		(* Ziel												UTF8->ASCII		BacNet Text		Textlistname									BacNet Funktion																BacNet Textlist type												TextId		*)	
		I_BO_3.sActiveText								:= 	fcUtfToAscii(	fcGetBcText(	GVL_BACNET.fbBacNetParameter.metGetTextListName(enTypeOfBacNetFunktionIn := enTypeOfBacNetFunktion.Type_Anlagefunktion,		enTypeOfBacNetTextListIn := enTypeOfBacNetTextList.PRESENTVALUE	),	'I_BO_3_ST_ACTIVE'		));
		I_BO_3.sInactiveText							:= 	fcUtfToAscii(	fcGetBcText(	GVL_BACNET.fbBacNetParameter.metGetTextListName(enTypeOfBacNetFunktionIn := enTypeOfBacNetFunktion.Type_Anlagefunktion,		enTypeOfBacNetTextListIn := enTypeOfBacNetTextList.PRESENTVALUE	),	'I_BO_3_ST_INACTIVE'	));	

		(* Ziel												Convert			BacNet Text		Textlistname									BacNet Funktion																BacNet Textlist type												TextId		*)	
		I_BO_3.udiNotificationClass						:= 	TO_UDINT	(	fcGetBcText(	GVL_BACNET.fbBacNetParameter.metGetTextListName(enTypeOfBacNetFunktionIn := enTypeOfBacNetFunktion.Type_Anlagefunktion,		enTypeOfBacNetTextListIn := enTypeOfBacNetTextList.NC			),	'I_BO_3_NC'	));	
		I_BO_3.eNotifyType								:= 	WagoTypesBACnet.eBACnetNotifyType.NOTIFY_TYPE_EVENT;
		
	ELSE
		I_BO_3.Delete();
	END_IF;
	(* Get Status *)
	metCreate_I_BO_3 := I_BO_3.xIsCreated;	
END_IF;
END_METHOD

METHOD metCreate_D_BV_4 : BOOL
(* D_BV_4*)
IF NOT D_BV_4.xIsCreated THEN
	(* Ziel						UTF8->ASCII						OBJ_NAME_BASE			BacNet Text		Textlistname									BacNet Funktion																BacNet Textlist type												TextId		*)
	D_BV_4._sObjectName		:=	fcUtfToAscii(Standard.CONCAT(	OBJ_NAME_BASE		,	fcGetBcText(	GVL_BACNET.fbBacNetParameter.metGetTextListName(enTypeOfBacNetFunktionIn := enTypeOfBacNetFunktion.Type_Anlagefunktion,		enTypeOfBacNetTextListIn := enTypeOfBacNetTextList.ENDING		),	'D_BV_4')));
	D_BV_4._sDescription	:= 	fcUtfToAscii(Standard.CONCAT(	OBJ_NAME_DESCRIPTION,	fcGetBcText(	GVL_BACNET.fbBacNetParameter.metGetTextListName(enTypeOfBacNetFunktionIn := enTypeOfBacNetFunktion.Type_Anlagefunktion,		enTypeOfBacNetTextListIn := enTypeOfBacNetTextList.DESCRIPTION	),	'D_BV_4')));
	(* Create Id from Base Id and Object Nr (Last nummber of Name *)	
	D_BV_4.Create(diInstance := TO_DINT(Standard.CONCAT(TO_STRING(dwOBJ_ID_BASE),'1')));
	(* Check if Created *)
	IF D_BV_4.xIsCreated THEN
		(* Set Group *)
		D_BV_4.setPropertyGroup(WagoTypesBacNet.eBACnetPropertyIdentifier.PROP_PRESENT_VALUE						,WagoTypesBacNet.eBACnetPropertyUpdateGroup.GROUP_CYCLIC);
		D_BV_4.setPropertyGroup(WagoTypesBacNet.eBACnetPropertyIdentifier.PROP_PRIORITY_ARRAY						,WagoTypesBacNet.eBACnetPropertyUpdateGroup.GROUP_CYCLIC);
		D_BV_4.setPropertyGroup(WagoTypesBacNet.eBACnetPropertyIdentifier.PROP_ELAPSED_ACTIVE_TIME					,WagoTypesBacNet.eBACnetPropertyUpdateGroup.GROUP_CYCLIC);
		D_BV_4.setPropertyGroup(WagoTypesBacNet.eBACnetPropertyIdentifier.PROP_DESCRIPTION							,WagoTypesBacNet.eBACnetPropertyUpdateGroup.GROUP_CYCLIC);
		D_BV_4.setPropertyGroup(WagoTypesBacNet.eBACnetPropertyIdentifier.PROP_EVENT_MESSAGE_TEXTS_CONFIG			,WagoTypesBacNet.eBACnetPropertyUpdateGroup.GROUP_CYCLIC);
			
		(* Ziel												UTF8->ASCII		BacNet Text		Textlistname									BacNet Funktion																BacNet Textlist type												TextId		*)
		D_BV_4.IEventMessageTextsConfig.sToOffNormal	:=	fcUtfToAscii(	fcGetBcText(	GVL_BACNET.fbBacNetParameter.metGetTextListName(enTypeOfBacNetFunktionIn := enTypeOfBacNetFunktion.Type_Anlagefunktion,		enTypeOfBacNetTextListIn := enTypeOfBacNetTextList.EVENTMESSAGE	),	'D_BV_4_ToOffNormal'	));		
		D_BV_4.IEventMessageTextsConfig.sToFault		:=	fcUtfToAscii(	fcGetBcText(	GVL_BACNET.fbBacNetParameter.metGetTextListName(enTypeOfBacNetFunktionIn := enTypeOfBacNetFunktion.Type_Anlagefunktion,		enTypeOfBacNetTextListIn := enTypeOfBacNetTextList.EVENTMESSAGE	),	'D_BV_4_ToFault'		));		
		D_BV_4.IEventMessageTextsConfig.sToNormal		:=	fcUtfToAscii(	fcGetBcText(	GVL_BACNET.fbBacNetParameter.metGetTextListName(enTypeOfBacNetFunktionIn := enTypeOfBacNetFunktion.Type_Anlagefunktion,		enTypeOfBacNetTextListIn := enTypeOfBacNetTextList.EVENTMESSAGE	),	'D_BV_4_ToNormal'		));		

		(* Ziel												UTF8->ASCII		BacNet Text		Textlistname									BacNet Funktion																BacNet Textlist type												TextId		*)	
		D_BV_4.sActiveText								:= 	fcUtfToAscii(	fcGetBcText(	GVL_BACNET.fbBacNetParameter.metGetTextListName(enTypeOfBacNetFunktionIn := enTypeOfBacNetFunktion.Type_Anlagefunktion,		enTypeOfBacNetTextListIn := enTypeOfBacNetTextList.PRESENTVALUE	),	'D_BV_4_ST_ACTIVE'		));
		D_BV_4.sInactiveText							:= 	fcUtfToAscii(	fcGetBcText(	GVL_BACNET.fbBacNetParameter.metGetTextListName(enTypeOfBacNetFunktionIn := enTypeOfBacNetFunktion.Type_Anlagefunktion,		enTypeOfBacNetTextListIn := enTypeOfBacNetTextList.PRESENTVALUE	),	'D_BV_4_ST_INACTIVE'	));	

		(* Ziel												Convert			BacNet Text		Textlistname									BacNet Funktion																BacNet Textlist type												TextId		*)	
		D_BV_4.udiNotificationClass						:= 	TO_UDINT	(	fcGetBcText(	GVL_BACNET.fbBacNetParameter.metGetTextListName(enTypeOfBacNetFunktionIn := enTypeOfBacNetFunktion.Type_Anlagefunktion,		enTypeOfBacNetTextListIn := enTypeOfBacNetTextList.NC			),	'D_BV_4_NC'	));	
		D_BV_4.eNotifyType								:= 	WagoTypesBACnet.eBACnetNotifyType.NOTIFY_TYPE_EVENT;
		D_BV_4.xAlarmValue								:= 	TO_BOOL		(	fcGetBcText(	GVL_BACNET.fbBacNetParameter.metGetTextListName(enTypeOfBacNetFunktionIn := enTypeOfBacNetFunktion.Type_Anlagefunktion,		enTypeOfBacNetTextListIn := enTypeOfBacNetTextList.NC		),	'D_BV_4_ALV'	));
	ELSE
		D_BV_4.Delete();
	END_IF;
	(* Get Status *)
	metCreate_D_BV_4 := D_BV_4.xIsCreated;	
END_IF;
END_METHOD

METHOD metCreate_E_BI_1 : BOOL
(* E_BI_1*)
IF NOT E_BI_1.xIsCreated THEN
	(* Ziel						UTF8->ASCII						OBJ_NAME_BASE			BacNet Text		Textlistname									BacNet Funktion																BacNet Textlist type												TextId		*)
	E_BI_1._sObjectName		:=	fcUtfToAscii(Standard.CONCAT(	OBJ_NAME_BASE		,	fcGetBcText(	GVL_BACNET.fbBacNetParameter.metGetTextListName(enTypeOfBacNetFunktionIn := enTypeOfBacNetFunktion.Type_Anlagefunktion,		enTypeOfBacNetTextListIn := enTypeOfBacNetTextList.ENDING		),	'E_BI_1')));
	E_BI_1._sDescription	:= 	fcUtfToAscii(Standard.CONCAT(	OBJ_NAME_DESCRIPTION,	fcGetBcText(	GVL_BACNET.fbBacNetParameter.metGetTextListName(enTypeOfBacNetFunktionIn := enTypeOfBacNetFunktion.Type_Anlagefunktion,		enTypeOfBacNetTextListIn := enTypeOfBacNetTextList.DESCRIPTION	),	'E_BI_1')));
	(* Create Id from Base Id and Object Nr (Last nummber of Name *)	
	E_BI_1.Create(diInstance := TO_DINT(Standard.CONCAT(TO_STRING(dwOBJ_ID_BASE),'1')));
	(* Check if Created *)
	IF E_BI_1.xIsCreated THEN
		(* Set Group *)
		E_BI_1.setPropertyGroup(WagoTypesBacNet.eBACnetPropertyIdentifier.PROP_PRESENT_VALUE						,WagoTypesBacNet.eBACnetPropertyUpdateGroup.GROUP_CYCLIC);
		E_BI_1.setPropertyGroup(WagoTypesBacNet.eBACnetPropertyIdentifier.PROP_PRIORITY_ARRAY						,WagoTypesBacNet.eBACnetPropertyUpdateGroup.GROUP_CYCLIC);
		E_BI_1.setPropertyGroup(WagoTypesBacNet.eBACnetPropertyIdentifier.PROP_ELAPSED_ACTIVE_TIME					,WagoTypesBacNet.eBACnetPropertyUpdateGroup.GROUP_CYCLIC);
		E_BI_1.setPropertyGroup(WagoTypesBacNet.eBACnetPropertyIdentifier.PROP_DESCRIPTION							,WagoTypesBacNet.eBACnetPropertyUpdateGroup.GROUP_CYCLIC);
		E_BI_1.setPropertyGroup(WagoTypesBacNet.eBACnetPropertyIdentifier.PROP_EVENT_MESSAGE_TEXTS_CONFIG			,WagoTypesBacNet.eBACnetPropertyUpdateGroup.GROUP_CYCLIC);
			
		(* Ziel												UTF8->ASCII		BacNet Text		Textlistname									BacNet Funktion																BacNet Textlist type												TextId		*)
		E_BI_1.IEventMessageTextsConfig.sToOffNormal	:=	fcUtfToAscii(	fcGetBcText(	GVL_BACNET.fbBacNetParameter.metGetTextListName(enTypeOfBacNetFunktionIn := enTypeOfBacNetFunktion.Type_Anlagefunktion,		enTypeOfBacNetTextListIn := enTypeOfBacNetTextList.EVENTMESSAGE	),	'E_BI_1_ToOffNormal'	));		
		E_BI_1.IEventMessageTextsConfig.sToFault		:=	fcUtfToAscii(	fcGetBcText(	GVL_BACNET.fbBacNetParameter.metGetTextListName(enTypeOfBacNetFunktionIn := enTypeOfBacNetFunktion.Type_Anlagefunktion,		enTypeOfBacNetTextListIn := enTypeOfBacNetTextList.EVENTMESSAGE	),	'E_BI_1_ToFault'		));		
		E_BI_1.IEventMessageTextsConfig.sToNormal		:=	fcUtfToAscii(	fcGetBcText(	GVL_BACNET.fbBacNetParameter.metGetTextListName(enTypeOfBacNetFunktionIn := enTypeOfBacNetFunktion.Type_Anlagefunktion,		enTypeOfBacNetTextListIn := enTypeOfBacNetTextList.EVENTMESSAGE	),	'E_BI_1_ToNormal'		));		

		(* Ziel												UTF8->ASCII		BacNet Text		Textlistname									BacNet Funktion																BacNet Textlist type												TextId		*)	
		E_BI_1.sActiveText								:= 	fcUtfToAscii(	fcGetBcText(	GVL_BACNET.fbBacNetParameter.metGetTextListName(enTypeOfBacNetFunktionIn := enTypeOfBacNetFunktion.Type_Anlagefunktion,		enTypeOfBacNetTextListIn := enTypeOfBacNetTextList.PRESENTVALUE	),	'E_BI_1_ST_ACTIVE'		));
		E_BI_1.sInactiveText							:= 	fcUtfToAscii(	fcGetBcText(	GVL_BACNET.fbBacNetParameter.metGetTextListName(enTypeOfBacNetFunktionIn := enTypeOfBacNetFunktion.Type_Anlagefunktion,		enTypeOfBacNetTextListIn := enTypeOfBacNetTextList.PRESENTVALUE	),	'E_BI_1_ST_INACTIVE'	));	

		(* Ziel												Convert			BacNet Text		Textlistname									BacNet Funktion																BacNet Textlist type												TextId		*)	
		E_BI_1.udiNotificationClass						:= 	TO_UDINT	(	fcGetBcText(	GVL_BACNET.fbBacNetParameter.metGetTextListName(enTypeOfBacNetFunktionIn := enTypeOfBacNetFunktion.Type_Anlagefunktion,		enTypeOfBacNetTextListIn := enTypeOfBacNetTextList.NC			),	'E_BI_1_NC'	));	
		E_BI_1.eNotifyType								:= 	WagoTypesBACnet.eBACnetNotifyType.NOTIFY_TYPE_EVENT;
		E_BI_1.xAlarmValue								:= 	TO_BOOL		(	fcGetBcText(	GVL_BACNET.fbBacNetParameter.metGetTextListName(enTypeOfBacNetFunktionIn := enTypeOfBacNetFunktion.Type_Anlagefunktion,		enTypeOfBacNetTextListIn := enTypeOfBacNetTextList.NC			),	'E_BI_1_ALV'	));
	ELSE
		E_BI_1.Delete();
	END_IF;
	(* Get Status *)
	metCreate_E_BI_1 := E_BI_1.xIsCreated;	
END_IF;
END_METHOD

METHOD metCreate_B_BV_2 : BOOL
(* B_BV_2*)
IF NOT B_BV_2.xIsCreated THEN
	(* Ziel						UTF8->ASCII						OBJ_NAME_BASE			BacNet Text		Textlistname									BacNet Funktion																BacNet Textlist type												TextId		*)
	B_BV_2._sObjectName		:=	fcUtfToAscii(Standard.CONCAT(	OBJ_NAME_BASE		,	fcGetBcText(	GVL_BACNET.fbBacNetParameter.metGetTextListName(enTypeOfBacNetFunktionIn := enTypeOfBacNetFunktion.Type_Anlagefunktion,		enTypeOfBacNetTextListIn := enTypeOfBacNetTextList.ENDING		),	'B_BV_2')));
	B_BV_2._sDescription	:= 	fcUtfToAscii(Standard.CONCAT(	OBJ_NAME_DESCRIPTION,	fcGetBcText(	GVL_BACNET.fbBacNetParameter.metGetTextListName(enTypeOfBacNetFunktionIn := enTypeOfBacNetFunktion.Type_Anlagefunktion,		enTypeOfBacNetTextListIn := enTypeOfBacNetTextList.DESCRIPTION	),	'B_BV_2')));
	(* Create Id from Base Id and Object Nr (Last nummber of Name *)	
	B_BV_2.Create(diInstance := TO_DINT(Standard.CONCAT(TO_STRING(dwOBJ_ID_BASE),'1')));
	(* Check if Created *)
	IF B_BV_2.xIsCreated THEN
		(* Set Group *)
		B_BV_2.setPropertyGroup(WagoTypesBacNet.eBACnetPropertyIdentifier.PROP_PRESENT_VALUE						,WagoTypesBacNet.eBACnetPropertyUpdateGroup.GROUP_CYCLIC);
		B_BV_2.setPropertyGroup(WagoTypesBacNet.eBACnetPropertyIdentifier.PROP_PRIORITY_ARRAY						,WagoTypesBacNet.eBACnetPropertyUpdateGroup.GROUP_CYCLIC);
		B_BV_2.setPropertyGroup(WagoTypesBacNet.eBACnetPropertyIdentifier.PROP_ELAPSED_ACTIVE_TIME					,WagoTypesBacNet.eBACnetPropertyUpdateGroup.GROUP_CYCLIC);
		B_BV_2.setPropertyGroup(WagoTypesBacNet.eBACnetPropertyIdentifier.PROP_DESCRIPTION							,WagoTypesBacNet.eBACnetPropertyUpdateGroup.GROUP_CYCLIC);
		B_BV_2.setPropertyGroup(WagoTypesBacNet.eBACnetPropertyIdentifier.PROP_EVENT_MESSAGE_TEXTS_CONFIG			,WagoTypesBacNet.eBACnetPropertyUpdateGroup.GROUP_CYCLIC);
			
		(* Ziel												UTF8->ASCII		BacNet Text		Textlistname									BacNet Funktion																BacNet Textlist type												TextId		*)
		B_BV_2.IEventMessageTextsConfig.sToOffNormal	:=	fcUtfToAscii(	fcGetBcText(	GVL_BACNET.fbBacNetParameter.metGetTextListName(enTypeOfBacNetFunktionIn := enTypeOfBacNetFunktion.Type_Anlagefunktion,		enTypeOfBacNetTextListIn := enTypeOfBacNetTextList.EVENTMESSAGE	),	'B_BV_2_ToOffNormal'	));		
		B_BV_2.IEventMessageTextsConfig.sToFault		:=	fcUtfToAscii(	fcGetBcText(	GVL_BACNET.fbBacNetParameter.metGetTextListName(enTypeOfBacNetFunktionIn := enTypeOfBacNetFunktion.Type_Anlagefunktion,		enTypeOfBacNetTextListIn := enTypeOfBacNetTextList.EVENTMESSAGE	),	'B_BV_2_ToFault'		));		
		B_BV_2.IEventMessageTextsConfig.sToNormal		:=	fcUtfToAscii(	fcGetBcText(	GVL_BACNET.fbBacNetParameter.metGetTextListName(enTypeOfBacNetFunktionIn := enTypeOfBacNetFunktion.Type_Anlagefunktion,		enTypeOfBacNetTextListIn := enTypeOfBacNetTextList.EVENTMESSAGE	),	'B_BV_2_ToNormal'		));		

		(* Ziel												UTF8->ASCII		BacNet Text		Textlistname									BacNet Funktion																BacNet Textlist type												TextId		*)	
		B_BV_2.sActiveText								:= 	fcUtfToAscii(	fcGetBcText(	GVL_BACNET.fbBacNetParameter.metGetTextListName(enTypeOfBacNetFunktionIn := enTypeOfBacNetFunktion.Type_Anlagefunktion,		enTypeOfBacNetTextListIn := enTypeOfBacNetTextList.PRESENTVALUE	),	'B_BV_2_ST_ACTIVE'		));
		B_BV_2.sInactiveText							:= 	fcUtfToAscii(	fcGetBcText(	GVL_BACNET.fbBacNetParameter.metGetTextListName(enTypeOfBacNetFunktionIn := enTypeOfBacNetFunktion.Type_Anlagefunktion,		enTypeOfBacNetTextListIn := enTypeOfBacNetTextList.PRESENTVALUE	),	'B_BV_2_ST_INACTIVE'	));	

		(* Ziel												Convert			BacNet Text		Textlistname									BacNet Funktion																BacNet Textlist type												TextId		*)	
		B_BV_2.udiNotificationClass						:= 	TO_UDINT	(	fcGetBcText(	GVL_BACNET.fbBacNetParameter.metGetTextListName(enTypeOfBacNetFunktionIn := enTypeOfBacNetFunktion.Type_Anlagefunktion,		enTypeOfBacNetTextListIn := enTypeOfBacNetTextList.NC			),	'B_BV_2_NC'	));	
		B_BV_2.eNotifyType								:= 	WagoTypesBACnet.eBACnetNotifyType.NOTIFY_TYPE_ALARM;
		B_BV_2.xAlarmValue								:= 	TO_BOOL		(	fcGetBcText(	GVL_BACNET.fbBacNetParameter.metGetTextListName(enTypeOfBacNetFunktionIn := enTypeOfBacNetFunktion.Type_Anlagefunktion,		enTypeOfBacNetTextListIn := enTypeOfBacNetTextList.NC		),	'B_BV_2_ALV'	));
		
	ELSE
		B_BV_2.Delete();
	END_IF;
	(* Get Status *)
	metCreate_B_BV_2 := B_BV_2.xIsCreated;	
END_IF;
END_METHOD

METHOD metCreate_C_BV_3 : BOOL
(* C_BV_3*)
IF NOT C_BV_3.xIsCreated THEN
	(* Ziel						UTF8->ASCII						OBJ_NAME_BASE			BacNet Text		Textlistname									BacNet Funktion																BacNet Textlist type												TextId		*)
	C_BV_3._sObjectName		:=	fcUtfToAscii(Standard.CONCAT(	OBJ_NAME_BASE		,	fcGetBcText(	GVL_BACNET.fbBacNetParameter.metGetTextListName(enTypeOfBacNetFunktionIn := enTypeOfBacNetFunktion.Type_Anlagefunktion,		enTypeOfBacNetTextListIn := enTypeOfBacNetTextList.ENDING		),	'C_BV_3')));
	C_BV_3._sDescription	:= 	fcUtfToAscii(Standard.CONCAT(	OBJ_NAME_DESCRIPTION,	fcGetBcText(	GVL_BACNET.fbBacNetParameter.metGetTextListName(enTypeOfBacNetFunktionIn := enTypeOfBacNetFunktion.Type_Anlagefunktion,		enTypeOfBacNetTextListIn := enTypeOfBacNetTextList.DESCRIPTION	),	'C_BV_3')));
	(* Create Id from Base Id and Object Nr (Last nummber of Name *)	
	C_BV_3.Create(diInstance := TO_DINT(Standard.CONCAT(TO_STRING(dwOBJ_ID_BASE),'1')));
	(* Check if Created *)
	IF C_BV_3.xIsCreated THEN
		(* Set Group *)
		C_BV_3.setPropertyGroup(WagoTypesBacNet.eBACnetPropertyIdentifier.PROP_PRESENT_VALUE						,WagoTypesBacNet.eBACnetPropertyUpdateGroup.GROUP_CYCLIC);
		C_BV_3.setPropertyGroup(WagoTypesBacNet.eBACnetPropertyIdentifier.PROP_PRIORITY_ARRAY						,WagoTypesBacNet.eBACnetPropertyUpdateGroup.GROUP_CYCLIC);
		C_BV_3.setPropertyGroup(WagoTypesBacNet.eBACnetPropertyIdentifier.PROP_ELAPSED_ACTIVE_TIME					,WagoTypesBacNet.eBACnetPropertyUpdateGroup.GROUP_CYCLIC);
		C_BV_3.setPropertyGroup(WagoTypesBacNet.eBACnetPropertyIdentifier.PROP_DESCRIPTION							,WagoTypesBacNet.eBACnetPropertyUpdateGroup.GROUP_CYCLIC);
		C_BV_3.setPropertyGroup(WagoTypesBacNet.eBACnetPropertyIdentifier.PROP_EVENT_MESSAGE_TEXTS_CONFIG			,WagoTypesBacNet.eBACnetPropertyUpdateGroup.GROUP_CYCLIC);
			
		(* Ziel												UTF8->ASCII		BacNet Text		Textlistname									BacNet Funktion																BacNet Textlist type												TextId		*)
		C_BV_3.IEventMessageTextsConfig.sToOffNormal	:=	fcUtfToAscii(	fcGetBcText(	GVL_BACNET.fbBacNetParameter.metGetTextListName(enTypeOfBacNetFunktionIn := enTypeOfBacNetFunktion.Type_Anlagefunktion,		enTypeOfBacNetTextListIn := enTypeOfBacNetTextList.EVENTMESSAGE	),	'C_BV_3_ToOffNormal'	));		
		C_BV_3.IEventMessageTextsConfig.sToFault		:=	fcUtfToAscii(	fcGetBcText(	GVL_BACNET.fbBacNetParameter.metGetTextListName(enTypeOfBacNetFunktionIn := enTypeOfBacNetFunktion.Type_Anlagefunktion,		enTypeOfBacNetTextListIn := enTypeOfBacNetTextList.EVENTMESSAGE	),	'C_BV_3_ToFault'		));		
		C_BV_3.IEventMessageTextsConfig.sToNormal		:=	fcUtfToAscii(	fcGetBcText(	GVL_BACNET.fbBacNetParameter.metGetTextListName(enTypeOfBacNetFunktionIn := enTypeOfBacNetFunktion.Type_Anlagefunktion,		enTypeOfBacNetTextListIn := enTypeOfBacNetTextList.EVENTMESSAGE	),	'C_BV_3_ToNormal'		));		

		(* Ziel												UTF8->ASCII		BacNet Text		Textlistname									BacNet Funktion																BacNet Textlist type												TextId		*)	
		C_BV_3.sActiveText								:= 	fcUtfToAscii(	fcGetBcText(	GVL_BACNET.fbBacNetParameter.metGetTextListName(enTypeOfBacNetFunktionIn := enTypeOfBacNetFunktion.Type_Anlagefunktion,		enTypeOfBacNetTextListIn := enTypeOfBacNetTextList.PRESENTVALUE	),	'C_BV_3_ST_ACTIVE'		));
		C_BV_3.sInactiveText							:= 	fcUtfToAscii(	fcGetBcText(	GVL_BACNET.fbBacNetParameter.metGetTextListName(enTypeOfBacNetFunktionIn := enTypeOfBacNetFunktion.Type_Anlagefunktion,		enTypeOfBacNetTextListIn := enTypeOfBacNetTextList.PRESENTVALUE	),	'C_BV_3_ST_INACTIVE'	));	

		(* Ziel												Convert			BacNet Text		Textlistname									BacNet Funktion																BacNet Textlist type												TextId		*)	
		C_BV_3.udiNotificationClass						:= 	TO_UDINT	(	fcGetBcText(	GVL_BACNET.fbBacNetParameter.metGetTextListName(enTypeOfBacNetFunktionIn := enTypeOfBacNetFunktion.Type_Anlagefunktion,		enTypeOfBacNetTextListIn := enTypeOfBacNetTextList.NC			),	'C_BV_3_NC'	));	
		C_BV_3.eNotifyType								:= 	WagoTypesBACnet.eBACnetNotifyType.NOTIFY_TYPE_ALARM;
		C_BV_3.xAlarmValue								:= 	TO_BOOL		(	fcGetBcText(	GVL_BACNET.fbBacNetParameter.metGetTextListName(enTypeOfBacNetFunktionIn := enTypeOfBacNetFunktion.Type_Anlagefunktion,		enTypeOfBacNetTextListIn := enTypeOfBacNetTextList.NC		),	'C_BV_3_ALV'	));
	ELSE
		C_BV_3.Delete();
	END_IF;
	(* Get Status *)
	metCreate_C_BV_3 := C_BV_3.xIsCreated;	
END_IF;
END_METHOD

METHOD metCreate_J_SC_1 : BOOL
(* J_SC_1*)
IF NOT J_SC_1.xIsCreated THEN
	(* Ziel						UTF8->ASCII						OBJ_NAME_BASE			BacNet Text		Textlistname									BacNet Funktion																BacNet Textlist type												TextId		*)
	J_SC_1._sObjectName		:=	fcUtfToAscii(Standard.CONCAT(	OBJ_NAME_BASE		,	fcGetBcText(	GVL_BACNET.fbBacNetParameter.metGetTextListName(enTypeOfBacNetFunktionIn := enTypeOfBacNetFunktion.Type_Anlagefunktion,		enTypeOfBacNetTextListIn := enTypeOfBacNetTextList.ENDING		),	'J_SC_1')));
	J_SC_1._sDescription	:= 	fcUtfToAscii(Standard.CONCAT(	OBJ_NAME_DESCRIPTION,	fcGetBcText(	GVL_BACNET.fbBacNetParameter.metGetTextListName(enTypeOfBacNetFunktionIn := enTypeOfBacNetFunktion.Type_Anlagefunktion,		enTypeOfBacNetTextListIn := enTypeOfBacNetTextList.DESCRIPTION	),	'J_SC_1')));
	(* Create Id from Base Id and Object Nr (Last nummber of Name *)	
	J_SC_1.Create(diInstance := TO_DINT(Standard.CONCAT(TO_STRING(dwOBJ_ID_BASE),'1')));
	(* Check if Created *)
	IF J_SC_1.xIsCreated THEN
		(* Set Group *)
		J_SC_1.setPropertyGroup(WagoTypesBacNet.eBACnetPropertyIdentifier.PROP_PRESENT_VALUE						,WagoTypesBacNet.eBACnetPropertyUpdateGroup.GROUP_CYCLIC);
		J_SC_1.setPropertyGroup(WagoTypesBacNet.eBACnetPropertyIdentifier.PROP_PRIORITY_ARRAY						,WagoTypesBacNet.eBACnetPropertyUpdateGroup.GROUP_CYCLIC);
		J_SC_1.setPropertyGroup(WagoTypesBacNet.eBACnetPropertyIdentifier.PROP_ELAPSED_ACTIVE_TIME					,WagoTypesBacNet.eBACnetPropertyUpdateGroup.GROUP_CYCLIC);
		J_SC_1.setPropertyGroup(WagoTypesBacNet.eBACnetPropertyIdentifier.PROP_DESCRIPTION							,WagoTypesBacNet.eBACnetPropertyUpdateGroup.GROUP_CYCLIC);
		J_SC_1.setPropertyGroup(WagoTypesBacNet.eBACnetPropertyIdentifier.PROP_EVENT_MESSAGE_TEXTS_CONFIG			,WagoTypesBacNet.eBACnetPropertyUpdateGroup.GROUP_CYCLIC);
			
		(* Ziel												UTF8->ASCII		BacNet Text		Textlistname									BacNet Funktion																BacNet Textlist type												TextId		*)
		J_SC_1.IEventMessageTextsConfig.sToOffNormal	:=	fcUtfToAscii(	fcGetBcText(	GVL_BACNET.fbBacNetParameter.metGetTextListName(enTypeOfBacNetFunktionIn := enTypeOfBacNetFunktion.Type_Anlagefunktion,		enTypeOfBacNetTextListIn := enTypeOfBacNetTextList.EVENTMESSAGE	),	'J_SC_1_ToOffNormal'	));		
		J_SC_1.IEventMessageTextsConfig.sToFault		:=	fcUtfToAscii(	fcGetBcText(	GVL_BACNET.fbBacNetParameter.metGetTextListName(enTypeOfBacNetFunktionIn := enTypeOfBacNetFunktion.Type_Anlagefunktion,		enTypeOfBacNetTextListIn := enTypeOfBacNetTextList.EVENTMESSAGE	),	'J_SC_1_ToFault'		));		
		J_SC_1.IEventMessageTextsConfig.sToNormal		:=	fcUtfToAscii(	fcGetBcText(	GVL_BACNET.fbBacNetParameter.metGetTextListName(enTypeOfBacNetFunktionIn := enTypeOfBacNetFunktion.Type_Anlagefunktion,		enTypeOfBacNetTextListIn := enTypeOfBacNetTextList.EVENTMESSAGE	),	'J_SC_1_ToNormal'		));		

		(* Ziel												Convert			BacNet Text		Textlistname									BacNet Funktion																BacNet Textlist type												TextId		*)	
		J_SC_1.udiNotificationClass						:= 	TO_UDINT	(	fcGetBcText(	GVL_BACNET.fbBacNetParameter.metGetTextListName(enTypeOfBacNetFunktionIn := enTypeOfBacNetFunktion.Type_Anlagefunktion,		enTypeOfBacNetTextListIn := enTypeOfBacNetTextList.NC			),	'J_SC_1_NC'	));	
		J_SC_1.eNotifyType								:= 	WagoTypesBACnet.eBACnetNotifyType.NOTIFY_TYPE_EVENT;
		
	ELSE
		J_SC_1.Delete();
	END_IF;
	(* Get Status *)
	metCreate_J_SC_1 := J_SC_1.xIsCreated;	
END_IF;
END_METHOD

METHOD metCreate_F_BV_5 : BOOL
(* F_BV_5*)
IF NOT F_BV_5.xIsCreated THEN
	(* Ziel						UTF8->ASCII						OBJ_NAME_BASE			BacNet Text		Textlistname									BacNet Funktion																BacNet Textlist type												TextId		*)
	F_BV_5._sObjectName		:=	fcUtfToAscii(Standard.CONCAT(	OBJ_NAME_BASE		,	fcGetBcText(	GVL_BACNET.fbBacNetParameter.metGetTextListName(enTypeOfBacNetFunktionIn := enTypeOfBacNetFunktion.Type_Anlagefunktion,		enTypeOfBacNetTextListIn := enTypeOfBacNetTextList.ENDING		),	'F_BV_5')));
	F_BV_5._sDescription	:= 	fcUtfToAscii(Standard.CONCAT(	OBJ_NAME_DESCRIPTION,	fcGetBcText(	GVL_BACNET.fbBacNetParameter.metGetTextListName(enTypeOfBacNetFunktionIn := enTypeOfBacNetFunktion.Type_Anlagefunktion,		enTypeOfBacNetTextListIn := enTypeOfBacNetTextList.DESCRIPTION	),	'F_BV_5')));
	(* Create Id from Base Id and Object Nr (Last nummber of Name *)	
	F_BV_5.Create(diInstance := TO_DINT(Standard.CONCAT(TO_STRING(dwOBJ_ID_BASE),'1')));
	(* Check if Created *)
	IF F_BV_5.xIsCreated THEN
		(* Set Group *)
		F_BV_5.setPropertyGroup(WagoTypesBacNet.eBACnetPropertyIdentifier.PROP_PRESENT_VALUE						,WagoTypesBacNet.eBACnetPropertyUpdateGroup.GROUP_CYCLIC);
		F_BV_5.setPropertyGroup(WagoTypesBacNet.eBACnetPropertyIdentifier.PROP_PRIORITY_ARRAY						,WagoTypesBacNet.eBACnetPropertyUpdateGroup.GROUP_CYCLIC);
		F_BV_5.setPropertyGroup(WagoTypesBacNet.eBACnetPropertyIdentifier.PROP_ELAPSED_ACTIVE_TIME					,WagoTypesBacNet.eBACnetPropertyUpdateGroup.GROUP_CYCLIC);
		F_BV_5.setPropertyGroup(WagoTypesBacNet.eBACnetPropertyIdentifier.PROP_DESCRIPTION							,WagoTypesBacNet.eBACnetPropertyUpdateGroup.GROUP_CYCLIC);
		F_BV_5.setPropertyGroup(WagoTypesBacNet.eBACnetPropertyIdentifier.PROP_EVENT_MESSAGE_TEXTS_CONFIG			,WagoTypesBacNet.eBACnetPropertyUpdateGroup.GROUP_CYCLIC);
			
		(* Ziel												UTF8->ASCII		BacNet Text		Textlistname									BacNet Funktion																BacNet Textlist type												TextId		*)
		F_BV_5.IEventMessageTextsConfig.sToOffNormal	:=	fcUtfToAscii(	fcGetBcText(	GVL_BACNET.fbBacNetParameter.metGetTextListName(enTypeOfBacNetFunktionIn := enTypeOfBacNetFunktion.Type_Anlagefunktion,		enTypeOfBacNetTextListIn := enTypeOfBacNetTextList.EVENTMESSAGE	),	'F_BV_5_ToOffNormal'	));		
		F_BV_5.IEventMessageTextsConfig.sToFault		:=	fcUtfToAscii(	fcGetBcText(	GVL_BACNET.fbBacNetParameter.metGetTextListName(enTypeOfBacNetFunktionIn := enTypeOfBacNetFunktion.Type_Anlagefunktion,		enTypeOfBacNetTextListIn := enTypeOfBacNetTextList.EVENTMESSAGE	),	'F_BV_5_ToFault'		));		
		F_BV_5.IEventMessageTextsConfig.sToNormal		:=	fcUtfToAscii(	fcGetBcText(	GVL_BACNET.fbBacNetParameter.metGetTextListName(enTypeOfBacNetFunktionIn := enTypeOfBacNetFunktion.Type_Anlagefunktion,		enTypeOfBacNetTextListIn := enTypeOfBacNetTextList.EVENTMESSAGE	),	'F_BV_5_ToNormal'		));		

		(* Ziel												UTF8->ASCII		BacNet Text		Textlistname									BacNet Funktion																BacNet Textlist type												TextId		*)	
		F_BV_5.sActiveText								:= 	fcUtfToAscii(	fcGetBcText(	GVL_BACNET.fbBacNetParameter.metGetTextListName(enTypeOfBacNetFunktionIn := enTypeOfBacNetFunktion.Type_Anlagefunktion,		enTypeOfBacNetTextListIn := enTypeOfBacNetTextList.PRESENTVALUE	),	'F_BV_5_ST_ACTIVE'		));
		F_BV_5.sInactiveText							:= 	fcUtfToAscii(	fcGetBcText(	GVL_BACNET.fbBacNetParameter.metGetTextListName(enTypeOfBacNetFunktionIn := enTypeOfBacNetFunktion.Type_Anlagefunktion,		enTypeOfBacNetTextListIn := enTypeOfBacNetTextList.PRESENTVALUE	),	'F_BV_5_ST_INACTIVE'	));	

		(* Ziel												Convert			BacNet Text		Textlistname									BacNet Funktion																BacNet Textlist type												TextId		*)	
		F_BV_5.udiNotificationClass						:= 	TO_UDINT	(	fcGetBcText(	GVL_BACNET.fbBacNetParameter.metGetTextListName(enTypeOfBacNetFunktionIn := enTypeOfBacNetFunktion.Type_Anlagefunktion,		enTypeOfBacNetTextListIn := enTypeOfBacNetTextList.NC			),	'F_BV_5_NC'	));	
		F_BV_5.eNotifyType								:= 	WagoTypesBACnet.eBACnetNotifyType.NOTIFY_TYPE_EVENT;
		F_BV_5.xAlarmValue								:= 	TO_BOOL		(	fcGetBcText(	GVL_BACNET.fbBacNetParameter.metGetTextListName(enTypeOfBacNetFunktionIn := enTypeOfBacNetFunktion.Type_Anlagefunktion,		enTypeOfBacNetTextListIn := enTypeOfBacNetTextList.NC			),	'F_BV_5_ALV'	));
		
	ELSE
		F_BV_5.Delete();
	END_IF;
	(* Get Status *)
	metCreate_F_BV_5 := F_BV_5.xIsCreated;	
END_IF;
END_METHOD

METHOD metCreate_G_BO_1 : BOOL
(* G_BO_1*)
IF NOT G_BO_1.xIsCreated THEN
	(* Ziel						UTF8->ASCII						OBJ_NAME_BASE			BacNet Text		Textlistname									BacNet Funktion																BacNet Textlist type												TextId		*)
	G_BO_1._sObjectName		:=	fcUtfToAscii(Standard.CONCAT(	OBJ_NAME_BASE		,	fcGetBcText(	GVL_BACNET.fbBacNetParameter.metGetTextListName(enTypeOfBacNetFunktionIn := enTypeOfBacNetFunktion.Type_Anlagefunktion,		enTypeOfBacNetTextListIn := enTypeOfBacNetTextList.ENDING		),	'G_BO_1')));
	G_BO_1._sDescription	:= 	fcUtfToAscii(Standard.CONCAT(	OBJ_NAME_DESCRIPTION,	fcGetBcText(	GVL_BACNET.fbBacNetParameter.metGetTextListName(enTypeOfBacNetFunktionIn := enTypeOfBacNetFunktion.Type_Anlagefunktion,		enTypeOfBacNetTextListIn := enTypeOfBacNetTextList.DESCRIPTION	),	'G_BO_1')));
	(* Create Id from Base Id and Object Nr (Last nummber of Name *)	
	G_BO_1.Create(diInstance := TO_DINT(Standard.CONCAT(TO_STRING(dwOBJ_ID_BASE),'1')));
	(* Check if Created *)
	IF G_BO_1.xIsCreated THEN
		(* Set Group *)
		G_BO_1.setPropertyGroup(WagoTypesBacNet.eBACnetPropertyIdentifier.PROP_PRESENT_VALUE						,WagoTypesBacNet.eBACnetPropertyUpdateGroup.GROUP_CYCLIC);
		G_BO_1.setPropertyGroup(WagoTypesBacNet.eBACnetPropertyIdentifier.PROP_PRIORITY_ARRAY						,WagoTypesBacNet.eBACnetPropertyUpdateGroup.GROUP_CYCLIC);
		G_BO_1.setPropertyGroup(WagoTypesBacNet.eBACnetPropertyIdentifier.PROP_ELAPSED_ACTIVE_TIME					,WagoTypesBacNet.eBACnetPropertyUpdateGroup.GROUP_CYCLIC);
		G_BO_1.setPropertyGroup(WagoTypesBacNet.eBACnetPropertyIdentifier.PROP_DESCRIPTION							,WagoTypesBacNet.eBACnetPropertyUpdateGroup.GROUP_CYCLIC);
		G_BO_1.setPropertyGroup(WagoTypesBacNet.eBACnetPropertyIdentifier.PROP_EVENT_MESSAGE_TEXTS_CONFIG			,WagoTypesBacNet.eBACnetPropertyUpdateGroup.GROUP_CYCLIC);
			
		(* Ziel												UTF8->ASCII		BacNet Text		Textlistname									BacNet Funktion																BacNet Textlist type												TextId		*)
		G_BO_1.IEventMessageTextsConfig.sToOffNormal	:=	fcUtfToAscii(	fcGetBcText(	GVL_BACNET.fbBacNetParameter.metGetTextListName(enTypeOfBacNetFunktionIn := enTypeOfBacNetFunktion.Type_Anlagefunktion,		enTypeOfBacNetTextListIn := enTypeOfBacNetTextList.EVENTMESSAGE	),	'G_BO_1_ToOffNormal'	));		
		G_BO_1.IEventMessageTextsConfig.sToFault		:=	fcUtfToAscii(	fcGetBcText(	GVL_BACNET.fbBacNetParameter.metGetTextListName(enTypeOfBacNetFunktionIn := enTypeOfBacNetFunktion.Type_Anlagefunktion,		enTypeOfBacNetTextListIn := enTypeOfBacNetTextList.EVENTMESSAGE	),	'G_BO_1_ToFault'		));		
		G_BO_1.IEventMessageTextsConfig.sToNormal		:=	fcUtfToAscii(	fcGetBcText(	GVL_BACNET.fbBacNetParameter.metGetTextListName(enTypeOfBacNetFunktionIn := enTypeOfBacNetFunktion.Type_Anlagefunktion,		enTypeOfBacNetTextListIn := enTypeOfBacNetTextList.EVENTMESSAGE	),	'G_BO_1_ToNormal'		));		

		(* Ziel												UTF8->ASCII		BacNet Text		Textlistname									BacNet Funktion																BacNet Textlist type												TextId		*)	
		G_BO_1.sActiveText								:= 	fcUtfToAscii(	fcGetBcText(	GVL_BACNET.fbBacNetParameter.metGetTextListName(enTypeOfBacNetFunktionIn := enTypeOfBacNetFunktion.Type_Anlagefunktion,		enTypeOfBacNetTextListIn := enTypeOfBacNetTextList.PRESENTVALUE	),	'G_BO_1_ST_ACTIVE'		));
		G_BO_1.sInactiveText							:= 	fcUtfToAscii(	fcGetBcText(	GVL_BACNET.fbBacNetParameter.metGetTextListName(enTypeOfBacNetFunktionIn := enTypeOfBacNetFunktion.Type_Anlagefunktion,		enTypeOfBacNetTextListIn := enTypeOfBacNetTextList.PRESENTVALUE	),	'G_BO_1_ST_INACTIVE'	));	

		(* Ziel												Convert			BacNet Text		Textlistname									BacNet Funktion																BacNet Textlist type												TextId		*)	
		G_BO_1.udiNotificationClass						:= 	TO_UDINT	(	fcGetBcText(	GVL_BACNET.fbBacNetParameter.metGetTextListName(enTypeOfBacNetFunktionIn := enTypeOfBacNetFunktion.Type_Anlagefunktion,		enTypeOfBacNetTextListIn := enTypeOfBacNetTextList.NC			),	'G_BO_1_NC'	));	
		G_BO_1.eNotifyType								:= 	WagoTypesBACnet.eBACnetNotifyType.NOTIFY_TYPE_EVENT;
		
	ELSE
		G_BO_1.Delete();
	END_IF;
	(* Get Status *)
	metCreate_G_BO_1 := G_BO_1.xIsCreated;	
END_IF;
END_METHOD

METHOD metCreate_A_BV_1 : BOOL
(* A_BV_1*)
IF NOT A_BV_1.xIsCreated THEN
	(* Ziel						UTF8->ASCII						OBJ_NAME_BASE			BacNet Text		Textlistname									BacNet Funktion																BacNet Textlist type												TextId		*)
	A_BV_1._sObjectName		:=	fcUtfToAscii(Standard.CONCAT(	OBJ_NAME_BASE		,	fcGetBcText(	GVL_BACNET.fbBacNetParameter.metGetTextListName(enTypeOfBacNetFunktionIn := enTypeOfBacNetFunktion.Type_Anlagefunktion,		enTypeOfBacNetTextListIn := enTypeOfBacNetTextList.ENDING		),	'A_BV_1')));
	A_BV_1._sDescription	:= 	fcUtfToAscii(Standard.CONCAT(	OBJ_NAME_DESCRIPTION,	fcGetBcText(	GVL_BACNET.fbBacNetParameter.metGetTextListName(enTypeOfBacNetFunktionIn := enTypeOfBacNetFunktion.Type_Anlagefunktion,		enTypeOfBacNetTextListIn := enTypeOfBacNetTextList.DESCRIPTION	),	'A_BV_1')));
	(* Create Id from Base Id and Object Nr (Last nummber of Name *)	
	A_BV_1.Create(diInstance := TO_DINT(Standard.CONCAT(TO_STRING(dwOBJ_ID_BASE),'1')));
	(* Check if Created *)
	IF A_BV_1.xIsCreated THEN
		(* Set Group *)
		A_BV_1.setPropertyGroup(WagoTypesBacNet.eBACnetPropertyIdentifier.PROP_PRESENT_VALUE						,WagoTypesBacNet.eBACnetPropertyUpdateGroup.GROUP_CYCLIC);
		A_BV_1.setPropertyGroup(WagoTypesBacNet.eBACnetPropertyIdentifier.PROP_PRIORITY_ARRAY						,WagoTypesBacNet.eBACnetPropertyUpdateGroup.GROUP_CYCLIC);
		A_BV_1.setPropertyGroup(WagoTypesBacNet.eBACnetPropertyIdentifier.PROP_ELAPSED_ACTIVE_TIME					,WagoTypesBacNet.eBACnetPropertyUpdateGroup.GROUP_CYCLIC);
		A_BV_1.setPropertyGroup(WagoTypesBacNet.eBACnetPropertyIdentifier.PROP_DESCRIPTION							,WagoTypesBacNet.eBACnetPropertyUpdateGroup.GROUP_CYCLIC);
		A_BV_1.setPropertyGroup(WagoTypesBacNet.eBACnetPropertyIdentifier.PROP_EVENT_MESSAGE_TEXTS_CONFIG			,WagoTypesBacNet.eBACnetPropertyUpdateGroup.GROUP_CYCLIC);
			
		(* Ziel												UTF8->ASCII		BacNet Text		Textlistname									BacNet Funktion																BacNet Textlist type												TextId		*)
		A_BV_1.IEventMessageTextsConfig.sToOffNormal	:=	fcUtfToAscii(	fcGetBcText(	GVL_BACNET.fbBacNetParameter.metGetTextListName(enTypeOfBacNetFunktionIn := enTypeOfBacNetFunktion.Type_Anlagefunktion,		enTypeOfBacNetTextListIn := enTypeOfBacNetTextList.EVENTMESSAGE	),	'A_BV_1_ToOffNormal'	));		
		A_BV_1.IEventMessageTextsConfig.sToFault		:=	fcUtfToAscii(	fcGetBcText(	GVL_BACNET.fbBacNetParameter.metGetTextListName(enTypeOfBacNetFunktionIn := enTypeOfBacNetFunktion.Type_Anlagefunktion,		enTypeOfBacNetTextListIn := enTypeOfBacNetTextList.EVENTMESSAGE	),	'A_BV_1_ToFault'		));		
		A_BV_1.IEventMessageTextsConfig.sToNormal		:=	fcUtfToAscii(	fcGetBcText(	GVL_BACNET.fbBacNetParameter.metGetTextListName(enTypeOfBacNetFunktionIn := enTypeOfBacNetFunktion.Type_Anlagefunktion,		enTypeOfBacNetTextListIn := enTypeOfBacNetTextList.EVENTMESSAGE	),	'A_BV_1_ToNormal'		));		

		(* Ziel												UTF8->ASCII		BacNet Text		Textlistname									BacNet Funktion																BacNet Textlist type												TextId		*)	
		A_BV_1.sActiveText								:= 	fcUtfToAscii(	fcGetBcText(	GVL_BACNET.fbBacNetParameter.metGetTextListName(enTypeOfBacNetFunktionIn := enTypeOfBacNetFunktion.Type_Anlagefunktion,		enTypeOfBacNetTextListIn := enTypeOfBacNetTextList.PRESENTVALUE	),	'A_BV_1_ST_ACTIVE'		));
		A_BV_1.sInactiveText							:= 	fcUtfToAscii(	fcGetBcText(	GVL_BACNET.fbBacNetParameter.metGetTextListName(enTypeOfBacNetFunktionIn := enTypeOfBacNetFunktion.Type_Anlagefunktion,		enTypeOfBacNetTextListIn := enTypeOfBacNetTextList.PRESENTVALUE	),	'A_BV_1_ST_INACTIVE'	));	

		(* Ziel												Convert			BacNet Text		Textlistname									BacNet Funktion																BacNet Textlist type												TextId		*)	
		A_BV_1.udiNotificationClass						:= 	TO_UDINT	(	fcGetBcText(	GVL_BACNET.fbBacNetParameter.metGetTextListName(enTypeOfBacNetFunktionIn := enTypeOfBacNetFunktion.Type_Anlagefunktion,		enTypeOfBacNetTextListIn := enTypeOfBacNetTextList.NC			),	'A_BV_1_NC'	));	
		A_BV_1.eNotifyType								:= 	WagoTypesBACnet.eBACnetNotifyType.NOTIFY_TYPE_ALARM;
		A_BV_1.xAlarmValue								:= 	TO_BOOL		(	fcGetBcText(	GVL_BACNET.fbBacNetParameter.metGetTextListName(enTypeOfBacNetFunktionIn := enTypeOfBacNetFunktion.Type_Anlagefunktion,		enTypeOfBacNetTextListIn := enTypeOfBacNetTextList.NC		),	'A_BV_1_ALV'	));
	ELSE
		A_BV_1.Delete();
	END_IF;
	(* Get Status *)
	metCreate_A_BV_1 := A_BV_1.xIsCreated;	
END_IF;
END_METHOD

METHOD metCREATE_KBOB_2017_V1 : BOOL;
VAR_INPUT
END_VAR
VAR
	oStatus		:	WagoSysErrorBase.FbResult;
	usiErrors	:	USINT;
END_VAR
(* Resett *)
usiErrors := 0;	

(* Create Objeccts *)
CASE usiCreateCase OF
	1:	
		usiErrors := usiErrors + TO_USINT(NOT metCreate_A_BV_1());
	2:
		usiErrors := usiErrors + TO_USINT(NOT metCreate_B_BV_2());
	3:	
		usiErrors := usiErrors + TO_USINT(NOT metCreate_C_BV_3());
	4:	
		usiErrors := usiErrors + TO_USINT(NOT metCreate_D_BV_4());
	5:
		usiErrors := usiErrors + TO_USINT(NOT metCreate_E_BI_1());
	6:	
		usiErrors := usiErrors + TO_USINT(NOT metCreate_F_BV_5());
	7:
		usiErrors := usiErrors + TO_USINT(NOT metCreate_G_BO_1());
	8:	
		usiErrors := usiErrors + TO_USINT(NOT metCreate_H_BO_2());
	9:
		usiErrors := usiErrors + TO_USINT(NOT metCreate_I_BO_3());
	10:
		usiErrors := usiErrors + TO_USINT(NOT metCreate_J_SC_1());
	0: 
		usiCreateCase := 1;
ELSE
	usiCreateCase := 0;
END_CASE;

(* STRUCT VIEW *)
metCREATE_STRUCTVIEW_KBOB_2017_V1();

(* OK = 0*)
metCREATE_KBOB_2017_V1 := NOT TO_BOOL(usiErrors);
END_METHOD

METHOD metCREATE_STRUCTVIEW_KBOB_2017_V1 : BOOL
VAR_INPUT
END_VAR
CASE usiCreateCase OF
	1:
		fcXMLStructuredView(THIS^,A_BV_1.IObjectIdentifier);
	2:
		fcXMLStructuredView(THIS^,B_BV_2.IObjectIdentifier);
	3:
		fcXMLStructuredView(THIS^,C_BV_3.IObjectIdentifier);
	4:
		fcXMLStructuredView(THIS^,D_BV_4.IObjectIdentifier);
	5:
		fcXMLStructuredView(THIS^,E_BI_1.IObjectIdentifier);
	6:
		fcXMLStructuredView(THIS^,F_BV_5.IObjectIdentifier);
	7:
		fcXMLStructuredView(THIS^,G_BO_1.IObjectIdentifier);
	8:
		fcXMLStructuredView(THIS^,H_BO_2.IObjectIdentifier);
	9:
		fcXMLStructuredView(THIS^,I_BO_3.IObjectIdentifier);
	10:
		fcXMLStructuredView(THIS^,J_SC_1.IObjectIdentifier);
		fcXMLAddStructuredViewToDevice(THIS^);	
	0: 
		usiCreateCase := 1;
ELSE
	usiCreateCase := 0;
END_CASE
END_METHOD

METHOD metCREATE : BOOL;
VAR_INPUT
END_VAR
VAR
	oStatus		:	WagoSysErrorBase.FbResult;
	usiErrors	:	USINT;
END_VAR
(* Get Revision *)
CASE GVL_BACNET.fbBacNetParameter.proKBOB_REV OF
	(* KBOB 2021 V2 *)
	enKBOB_REV.KBOB_REV2021_V2:
		usiErrors := usiErrors + TO_USINT(NOT metCREATE_KBOB_2021_V2());
	(* KBOB 2017 V1 *)
	enKBOB_REV.KBOB_REV2017_V1:
		usiErrors := usiErrors + TO_USINT(NOT metCREATE_KBOB_2017_V1());
	(* Default *)
	ELSE
		usiErrors := usiErrors + TO_USINT(NOT metCREATE_KBOB_2021_V2());
END_CASE;

(* OK = 0*)
xErrorCreate := TO_BOOL(usiErrors);
metCREATE := NOT TO_BOOL(usiErrors) AND usiCreateCase = usiAnzBacNetObj;
END_METHOD

METHOD metCYCLIC_KBOB_2017_V1
VAR_INPUT
END_VAR
(* A_BV_1 Objektschutz *)
IF A_BV_1.xIsCreated THEN
	IF A_BV_1.xPresentValue <> xObjektSchutz THEN
		A_BV_1.xPresentValue := xObjektSchutz;
	END_IF;
END_IF;

(* B_BV_2 Technischer Alarm *)
IF B_BV_2.xIsCreated THEN
	IF B_BV_2.xPresentValue <> xTechnischerAlarm THEN
		B_BV_2.xPresentValue := xTechnischerAlarm;
	END_IF;
END_IF;

(* C_BV_3 Technischer Störung *)
IF C_BV_3.xIsCreated THEN
	IF C_BV_3.xPresentValue <> xTechnischeStörung THEN
		C_BV_3.xPresentValue := xTechnischeStörung;
	END_IF;
END_IF;

(* D_BV_4 Wartungsmeldung *)
IF D_BV_4.xIsCreated THEN
	IF D_BV_4.xPresentValue <> xWartungsmeldung THEN
		D_BV_4.xPresentValue := xWartungsmeldung;
	END_IF;
END_IF;

(* E_BI_1 Bedienung Lokal *)
IF E_BI_1.xIsCreated THEN
	IF E_BI_1.xPresentValue <> xBedienungLokal THEN
		E_BI_1.xPresentValue := xBedienungLokal;
	END_IF;
END_IF;

(* F_BV_5 Alarmunterdrückung *)
IF E_BI_1.xIsCreated THEN
	IF E_BI_1.xPresentValue <> xAlarmUnterdrückung THEN
		E_BI_1.xPresentValue := xAlarmUnterdrückung;
	END_IF;
END_IF;

(* G_BO_1 Signalisation Betrieb *)
IF G_BO_1.xIsCreated THEN
	IF G_BO_1.xPresentValue <> xAcknowledge THEN
		G_BO_1.xPresentValue := xAcknowledge;
	END_IF;
END_IF;

(* H_BO_2 Signalisation Sammelalarm *)
IF H_BO_2.xIsCreated THEN
	H_BO_2.xPresentValue := xObjektSchutz OR xTechnischerAlarm OR xTechnischeStörung ;
END_IF;

(* I_BO_3 Signalisation Bedienung Lokal *)
IF I_BO_3.xIsCreated THEN
	IF I_BO_3.xPresentValue <> xBedienungLokal THEN
		I_BO_3.xPresentValue := xBedienungLokal;
	END_IF;
END_IF;

(* I_BO_3 Zeitschaltuhr *)
IF J_SC_1.xIsCreated THEN
	IF J_SC_1.IPresentValue.eDataType = WagoTypesBACnet.eBACnetDataType.BACNET_TYPE_BOOLEAN THEN
		xZeitschaltUhr := J_SC_1.IPresentValue.IBOOL.xValue;
	END_IF;
END_IF;
END_METHOD

METHOD metCYCLIC_KBOB_2021_V2
VAR_INPUT
END_VAR
(* A_BV_1 Objektschutz *)
IF A_BV_1.xIsCreated THEN
	IF A_BV_1.xPresentValue <> xObjektSchutz THEN
		A_BV_1.xPresentValue := xObjektSchutz;
	END_IF;
END_IF;

(* B_BV_2 Technischer Alarm *)
IF B_BV_2.xIsCreated THEN
	IF B_BV_2.xPresentValue <> xTechnischerAlarm THEN
		B_BV_2.xPresentValue := xTechnischerAlarm;
	END_IF;
END_IF;

(* C_BV_3 Technischer Störung *)
IF C_BV_3.xIsCreated THEN
	IF C_BV_3.xPresentValue <> xTechnischeStörung THEN
		C_BV_3.xPresentValue := xTechnischeStörung;
	END_IF;
END_IF;

(* D_BV_4 Wartungsmeldung *)
IF D_BV_4.xIsCreated THEN
	IF D_BV_4.xPresentValue <> xWartungsmeldung THEN
		D_BV_4.xPresentValue := xWartungsmeldung;
	END_IF;
END_IF;

(* E_BI_1 Bedienung Lokal *)
IF E_BI_1.xIsCreated THEN
	IF E_BI_1.xPresentValue <> xBedienungLokal THEN
		E_BI_1.xPresentValue := xBedienungLokal;
	END_IF;
END_IF;

(* F_BV_5 Alarmunterdrückung *)
IF E_BI_1.xIsCreated THEN
	IF E_BI_1.xPresentValue <> xAlarmUnterdrückung THEN
		E_BI_1.xPresentValue := xAlarmUnterdrückung;
	END_IF;
END_IF;

(* G_BO_1 Signalisation Betrieb *)
IF G_BO_1.xIsCreated THEN
	IF G_BO_1.xPresentValue <> xAcknowledge THEN
		G_BO_1.xPresentValue := xAcknowledge;
	END_IF;
END_IF;

(* H_BO_2 Signalisation Sammelalarm *)
IF H_BO_2.xIsCreated THEN
	H_BO_2.xPresentValue := xObjektSchutz OR xTechnischerAlarm OR xTechnischeStörung ;
END_IF;

(* I_BO_3 Signalisation Bedienung Lokal *)
IF I_BO_3.xIsCreated THEN
	IF I_BO_3.xPresentValue <> xBedienungLokal THEN
		I_BO_3.xPresentValue := xBedienungLokal;
	END_IF;
END_IF;

(* I_BO_3 Zeitschaltuhr *)
IF J_SC_1.xIsCreated THEN
	IF J_SC_1.IPresentValue.eDataType = WagoTypesBACnet.eBACnetDataType.BACNET_TYPE_BOOLEAN THEN
		xZeitschaltUhr := J_SC_1.IPresentValue.IBOOL.xValue;
	END_IF;
END_IF;
END_METHOD

METHOD metCYCLIC_DESCRIPTION_FIX
VAR_INPUT
END_VAR
(* A_BO_1 *)
IF A_BV_1.xIsCreated THEN
	IF A_BV_1.sDescription <> A_BV_1._sDescription THEN
		A_BV_1.sDescription := A_BV_1._sDescription;
	END_IF;
END_IF;

(* B_BV_2 *)
IF B_BV_2.xIsCreated THEN
	IF B_BV_2.sDescription <> B_BV_2._sDescription THEN
		B_BV_2.sDescription := B_BV_2._sDescription;
	END_IF;
END_IF;

(* C_BV_3 *)
IF C_BV_3.xIsCreated THEN
	IF C_BV_3.sDescription <> C_BV_3._sDescription THEN
		C_BV_3.sDescription := C_BV_3._sDescription;
	END_IF;
END_IF;

(* D_BV_4 *)
IF D_BV_4.xIsCreated THEN
	IF D_BV_4.sDescription <> D_BV_4._sDescription THEN
		D_BV_4.sDescription := D_BV_4._sDescription;
	END_IF;
END_IF;

(* E_BI_1 *)
IF E_BI_1.xIsCreated THEN
	IF E_BI_1.sDescription <> E_BI_1._sDescription THEN
		E_BI_1.sDescription := E_BI_1._sDescription;
	END_IF;
END_IF;

(* F_BV_5 *)
IF F_BV_5.xIsCreated THEN
	IF F_BV_5.sDescription <> F_BV_5._sDescription THEN
		F_BV_5.sDescription := F_BV_5._sDescription;
	END_IF;
END_IF;

(* G_BO_1 *)
IF G_BO_1.xIsCreated THEN
	IF G_BO_1.sDescription <> G_BO_1._sDescription THEN
		G_BO_1.sDescription := G_BO_1._sDescription;
	END_IF;
END_IF;

(* H_BO_2 *)
IF H_BO_2.xIsCreated THEN
	IF H_BO_2.sDescription <> H_BO_2._sDescription THEN
		H_BO_2.sDescription := H_BO_2._sDescription;
	END_IF;
END_IF;

(* I_BO_3 *)
IF I_BO_3.xIsCreated THEN
	IF I_BO_3.sDescription <> I_BO_3._sDescription THEN
		I_BO_3.sDescription := I_BO_3._sDescription;
	END_IF;
END_IF;

(* J_SC_1 *)
IF J_SC_1.xIsCreated THEN
	IF J_SC_1.sDescription <> J_SC_1._sDescription THEN
		J_SC_1.sDescription := J_SC_1._sDescription;
	END_IF;
END_IF;
END_METHOD

(*FB_Exit muss explizit implementiert werden. Wenn es eine Implementierung gibt, dann wird 
die Methode aufgerufen, bevor die Steuerung den Code der Funktionsbaustein-Instanz entfernt
(impliziter Aufruf. Der Rückgabewert wird nicht ausgewertet.*)
METHOD FB_Exit : BOOL
VAR_INPUT
	(* TRUE: Die Exit-Methode wird aufgerufen, um die Instanz zu verlassen, die hinterher kopiert wird Online-Change).  *)
	bInCopyCode	: BOOL;
END_VAR
(* A_BV_1*)
IF A_BV_1.xIsCreated THEN
	A_BV_1.Delete();
END_IF;	
(* B_BV_2 *)
IF B_BV_2.xIsCreated THEN
	B_BV_2.Delete();
END_IF;	
(* C_BV_3 *)
IF C_BV_3.xIsCreated THEN
	C_BV_3.Delete();
END_IF;
(* D_BV_4 *)
IF D_BV_4.xIsCreated THEN
	D_BV_4.Delete();
END_IF;
(* E_BI_1 *)
IF E_BI_1.xIsCreated THEN
	E_BI_1.Delete();	
END_IF;
(* F_BV_5 *)
IF F_BV_5.xIsCreated THEN
	F_BV_5.Delete();
END_IF;
(* G_BO_1 *)
IF G_BO_1.xIsCreated THEN
	G_BO_1.Delete();
END_IF;
(* H_BO_2 *)
IF H_BO_2.xIsCreated THEN
	H_BO_2.Delete();
END_IF;
(* I_BO_3 *)
IF I_BO_3.xIsCreated THEN
	I_BO_3.Delete();
END_IF;
(* J_SC_1 *)
IF J_SC_1.xIsCreated THEN
	J_SC_1.Delete();
END_IF;
END_METHOD

METHOD metDELETE : BOOL
VAR_INPUT
END_VAR
(* A_BV_1*)
IF A_BV_1.xIsCreated THEN
	A_BV_1.Delete();
END_IF;	
(* B_BV_2 *)
IF B_BV_2.xIsCreated THEN
	B_BV_2.Delete();
END_IF;	
(* C_BV_3 *)
IF C_BV_3.xIsCreated THEN
	C_BV_3.Delete();
END_IF;
(* D_BV_4 *)
IF D_BV_4.xIsCreated THEN
	D_BV_4.Delete();
END_IF;
(* E_BI_1 *)
IF E_BI_1.xIsCreated THEN
	E_BI_1.Delete();	
END_IF;
(* F_BV_5 *)
IF F_BV_5.xIsCreated THEN
	F_BV_5.Delete();
END_IF;
(* G_BO_1 *)
IF G_BO_1.xIsCreated THEN
	G_BO_1.Delete();
END_IF;
(* H_BO_2 *)
IF H_BO_2.xIsCreated THEN
	H_BO_2.Delete();
END_IF;
(* I_BO_3 *)
IF I_BO_3.xIsCreated THEN
	I_BO_3.Delete();
END_IF;
(* J_SC_1 *)
IF J_SC_1.xIsCreated THEN
	J_SC_1.Delete();
END_IF;

(* Delete Struct View *)
IF GVL_BACNET.fbBacNetParameter.proDestroyBacNetOverrideXmlNode THEN
	fcXMLDeleteOverrideNode(fcBacNetIdToIdWitType(TO_DINT(CONCAT(TO_STRING(OBJ_ID_BASE),'1')),WagoTypesBacNet.eBACnetObjectType.BACnet_structured_view));
	fcXMLDeleteStructuredViewFromDevice(fcBacNetIdToIdWitType(TO_DINT(CONCAT(TO_STRING(OBJ_ID_BASE),'1')),WagoTypesBacNet.eBACnetObjectType.BACnet_structured_view));
END_IF;

metDELETE := 	A_BV_1.xIsCreated OR 
				B_BV_2.xIsCreated OR
				C_BV_3.xIsCreated OR				
				D_BV_4.xIsCreated OR
				E_BI_1.xIsCreated OR
				F_BV_5.xIsCreated OR
				G_BO_1.xIsCreated OR
				H_BO_2.xIsCreated OR
				I_BO_3.xIsCreated OR
				J_SC_1.xIsCreated;
				
				
				
(* Reset Create Case *)
usiCreateCase := 1;
END_METHOD

END_FUNCTION_BLOCK

// 30 Program Organization Units/FBs/AT_FUNKTIONEN/AT_ZÄHLER/FB_AT_ZÄHLER
FUNCTION_BLOCK FB_AT_ZÄHLER EXTENDS FB_OBJ_ID_BASE
VAR_INPUT
	rValue				:	REAL;
	xError				:	BOOL;
END_VAR
VAR_OUTPUT

END_VAR
VAR
	(* BacNet Objects *)
	A_AV_1		:	WagoSysBACnet.FbAnalogValue_large(-1);					// Messwert
	B_TL_1		:	WagoSysBACnet.FbTrendLog_large(-1);                     // Aufzeichnung Messwert
	C_BV_1		:	WagoSysBACnet.FbBinaryValue_large(-1);              	// Störung

END_VAR
VAR CONSTANT
	usiAnzBacNetObj	:	USINT	:= 3;
END_VAR

(* Call Base FB*)
SUPER^();
(* Cyclic Action *)
IF xCreatet THEN
	(* DESCTIPTION FIX *)
	metCYCLIC_DESCRIPTION_FIX();
	(* Get Revision *)
	CASE GVL_BACNET.fbBacNetParameter.proKBOB_REV OF
		(* KBOB 2021 V2 *)
		enKBOB_REV.KBOB_REV2021_V2:
			metCYCLIC_KBOB_2021_V2();
		(* KBOB 2017 V1 *)
		enKBOB_REV.KBOB_REV2017_V1:
			metCYCLIC_KBOB_2017_V1();
		(* Default *)
		ELSE
			metCYCLIC_KBOB_2021_V2();
	END_CASE;	
END_IF;

METHOD metCREATE_STRUCTVIEW_KBOB_2021_V2 : BOOL
VAR_INPUT
END_VAR
CASE usiCreateCase OF
	1:	
		fcXMLStructuredView(THIS^,A_AV_1.IObjectIdentifier);
	2:
		fcXMLStructuredView(THIS^,B_TL_1.IObjectIdentifier);
	3:
		fcXMLStructuredView(THIS^,C_BV_1.IObjectIdentifier);
		fcXMLAddStructuredViewToDevice(THIS^);
	0: 
		usiCreateCase := 1;
ELSE
	usiCreateCase := 0;
END_CASE
END_METHOD

METHOD metCREATE_KBOB_2021_V2 : BOOL;
VAR_INPUT
END_VAR
VAR
	oStatus		:	WagoSysErrorBase.FbResult;
	usiErrors	:	USINT;
END_VAR
(* Resett *)
usiErrors := 0;	

(* Create Objeccts *)
CASE usiCreateCase OF
	1:	
		usiErrors := usiErrors + TO_USINT(NOT metCreate_A_AV_1());
	2:
		usiErrors := usiErrors + TO_USINT(NOT metCreate_B_TL_1());
	3:	
		usiErrors := usiErrors + TO_USINT(NOT metCreate_C_BV_1());
	0: 
		usiCreateCase := 1;
ELSE
	usiCreateCase := 0;
END_CASE;

(* STRUCT VIEW *)
metCREATE_STRUCTVIEW_KBOB_2021_V2();

(* OK = 0*)
metCREATE_KBOB_2021_V2 := NOT TO_BOOL(usiErrors);
END_METHOD

METHOD metCreate_A_AV_1 : BOOL
(* A_AV_1*)
IF NOT A_AV_1.xIsCreated THEN
	(* Ziel						UTF8->ASCII						OBJ_NAME_BASE			BacNet Text		Textlistname									BacNet Funktion																	BacNet Textlist type												TextId		*)
	A_AV_1._sObjectName		:=	fcUtfToAscii(Standard.CONCAT(	OBJ_NAME_BASE		,	fcGetBcText(	GVL_BACNET.fbBacNetParameter.metGetTextListName(enTypeOfBacNetFunktionIn := enTypeOfBacNetFunktion.Type_Zähler,		enTypeOfBacNetTextListIn := enTypeOfBacNetTextList.ENDING		),	'A_AV_1')));
	A_AV_1._sDescription	:= 	fcUtfToAscii(Standard.CONCAT(	OBJ_NAME_DESCRIPTION,	fcGetBcText(	GVL_BACNET.fbBacNetParameter.metGetTextListName(enTypeOfBacNetFunktionIn := enTypeOfBacNetFunktion.Type_Zähler,		enTypeOfBacNetTextListIn := enTypeOfBacNetTextList.DESCRIPTION	),	'A_AV_1')));
	(* Create Id from Base Id and Object Nr (Last nummber of Name *)	
	A_AV_1.Create(diInstance := TO_DINT(Standard.CONCAT(TO_STRING(dwOBJ_ID_BASE),'1')));
	(* Check if Created *)
	IF A_AV_1.xIsCreated THEN
		(* Set Group *)
		A_AV_1.setPropertyGroup(WagoTypesBacNet.eBACnetPropertyIdentifier.PROP_PRESENT_VALUE						,WagoTypesBacNet.eBACnetPropertyUpdateGroup.GROUP_CYCLIC);
		A_AV_1.setPropertyGroup(WagoTypesBacNet.eBACnetPropertyIdentifier.PROP_PRIORITY_ARRAY						,WagoTypesBacNet.eBACnetPropertyUpdateGroup.GROUP_CYCLIC);
		A_AV_1.setPropertyGroup(WagoTypesBacNet.eBACnetPropertyIdentifier.PROP_ELAPSED_ACTIVE_TIME					,WagoTypesBacNet.eBACnetPropertyUpdateGroup.GROUP_CYCLIC);
		A_AV_1.setPropertyGroup(WagoTypesBacNet.eBACnetPropertyIdentifier.PROP_DESCRIPTION							,WagoTypesBacNet.eBACnetPropertyUpdateGroup.GROUP_CYCLIC);
		A_AV_1.setPropertyGroup(WagoTypesBacNet.eBACnetPropertyIdentifier.PROP_EVENT_MESSAGE_TEXTS_CONFIG			,WagoTypesBacNet.eBACnetPropertyUpdateGroup.GROUP_CYCLIC);
		(* Set Description to Overwrite retain*)
		A_AV_1.sDescription	:= A_AV_1._sDescription;
		(* Ziel												UTF8->ASCII		BacNet Text		Textlistname									BacNet Funktion																	BacNet Textlist type												TextId		*)
		A_AV_1.IEventMessageTextsConfig.sToOffNormal	:=	fcUtfToAscii(	fcGetBcText(	GVL_BACNET.fbBacNetParameter.metGetTextListName(enTypeOfBacNetFunktionIn := enTypeOfBacNetFunktion.Type_Zähler,		enTypeOfBacNetTextListIn := enTypeOfBacNetTextList.EVENTMESSAGE	),	'A_AV_1_ToOffNormal'	));		
		A_AV_1.IEventMessageTextsConfig.sToFault		:=	fcUtfToAscii(	fcGetBcText(	GVL_BACNET.fbBacNetParameter.metGetTextListName(enTypeOfBacNetFunktionIn := enTypeOfBacNetFunktion.Type_Zähler,		enTypeOfBacNetTextListIn := enTypeOfBacNetTextList.EVENTMESSAGE	),	'A_AV_1_ToFault'		));		
		A_AV_1.IEventMessageTextsConfig.sToNormal		:=	fcUtfToAscii(	fcGetBcText(	GVL_BACNET.fbBacNetParameter.metGetTextListName(enTypeOfBacNetFunktionIn := enTypeOfBacNetFunktion.Type_Zähler,		enTypeOfBacNetTextListIn := enTypeOfBacNetTextList.EVENTMESSAGE	),	'A_AV_1_ToNormal'		));		

		(* Ziel												Convert			BacNet Text		Textlistname									BacNet Funktion																	BacNet Textlist type												TextId		*)	
		A_AV_1.udiNotificationClass						:= 	TO_UDINT	(	fcGetBcText(	GVL_BACNET.fbBacNetParameter.metGetTextListName(enTypeOfBacNetFunktionIn := enTypeOfBacNetFunktion.Type_Zähler,		enTypeOfBacNetTextListIn := enTypeOfBacNetTextList.NC			),	'A_AV_1_NC'	));	
		A_AV_1.eNotifyType								:= 	WagoTypesBACnet.eBACnetNotifyType.NOTIFY_TYPE_EVENT;
		
	ELSE
		A_AV_1.Delete();
	END_IF;
	(* Get Status *)
	metCreate_A_AV_1 := A_AV_1.xIsCreated;	
END_IF;
END_METHOD

METHOD metCreate_B_TL_1 : BOOL
(* B_TL_1*)
IF NOT B_TL_1.xIsCreated THEN
	(* Ziel						UTF8->ASCII						OBJ_NAME_BASE			BacNet Text		Textlistname									BacNet Funktion																BacNet Textlist type												TextId		*)
	B_TL_1._sObjectName		:=	fcUtfToAscii(Standard.CONCAT(	OBJ_NAME_BASE		,	fcGetBcText(	GVL_BACNET.fbBacNetParameter.metGetTextListName(enTypeOfBacNetFunktionIn := enTypeOfBacNetFunktion.Type_Zähler,		enTypeOfBacNetTextListIn := enTypeOfBacNetTextList.ENDING		),	'B_TL_1')));
	B_TL_1._sDescription	:= 	fcUtfToAscii(Standard.CONCAT(	OBJ_NAME_DESCRIPTION,	fcGetBcText(	GVL_BACNET.fbBacNetParameter.metGetTextListName(enTypeOfBacNetFunktionIn := enTypeOfBacNetFunktion.Type_Zähler,		enTypeOfBacNetTextListIn := enTypeOfBacNetTextList.DESCRIPTION	),	'B_TL_1')));
	(* Create Id from Base Id and Object Nr (Last nummber of Name *)	
	B_TL_1.Create(diInstance := TO_DINT(Standard.CONCAT(TO_STRING(dwOBJ_ID_BASE),'1')));
	(* Check if Created *)
	IF B_TL_1.xIsCreated THEN
		(* Set Group *)
		B_TL_1.setPropertyGroup(WagoTypesBacNet.eBACnetPropertyIdentifier.PROP_PRESENT_VALUE						,WagoTypesBacNet.eBACnetPropertyUpdateGroup.GROUP_CYCLIC);
		B_TL_1.setPropertyGroup(WagoTypesBacNet.eBACnetPropertyIdentifier.PROP_PRIORITY_ARRAY						,WagoTypesBacNet.eBACnetPropertyUpdateGroup.GROUP_CYCLIC);
		B_TL_1.setPropertyGroup(WagoTypesBacNet.eBACnetPropertyIdentifier.PROP_ELAPSED_ACTIVE_TIME					,WagoTypesBacNet.eBACnetPropertyUpdateGroup.GROUP_CYCLIC);
		B_TL_1.setPropertyGroup(WagoTypesBacNet.eBACnetPropertyIdentifier.PROP_DESCRIPTION							,WagoTypesBacNet.eBACnetPropertyUpdateGroup.GROUP_CYCLIC);
		B_TL_1.setPropertyGroup(WagoTypesBacNet.eBACnetPropertyIdentifier.PROP_EVENT_MESSAGE_TEXTS_CONFIG			,WagoTypesBacNet.eBACnetPropertyUpdateGroup.GROUP_CYCLIC);
		(* Crate Override *)
		fcXMLTrendLogOverride(B_TL_1,A_AV_1.IObjectIdentifier,WagoTypesBacNet.eBACnetPropertyIdentifier.PROP_PRESENT_VALUE);
		(* Set Description to Overwrite retain*)
		B_TL_1.sDescription	:= B_TL_1._sDescription;
		(* Ziel												UTF8->ASCII		BacNet Text		Textlistname									BacNet Funktion																BacNet Textlist type												TextId		*)
		B_TL_1.IEventMessageTextsConfig.sToOffNormal	:=	fcUtfToAscii(	fcGetBcText(	GVL_BACNET.fbBacNetParameter.metGetTextListName(enTypeOfBacNetFunktionIn := enTypeOfBacNetFunktion.Type_Zähler,		enTypeOfBacNetTextListIn := enTypeOfBacNetTextList.EVENTMESSAGE	),	'B_TL_1_ToOffNormal'	));		
		B_TL_1.IEventMessageTextsConfig.sToFault		:=	fcUtfToAscii(	fcGetBcText(	GVL_BACNET.fbBacNetParameter.metGetTextListName(enTypeOfBacNetFunktionIn := enTypeOfBacNetFunktion.Type_Zähler,		enTypeOfBacNetTextListIn := enTypeOfBacNetTextList.EVENTMESSAGE	),	'B_TL_1_ToFault'		));		
		B_TL_1.IEventMessageTextsConfig.sToNormal		:=	fcUtfToAscii(	fcGetBcText(	GVL_BACNET.fbBacNetParameter.metGetTextListName(enTypeOfBacNetFunktionIn := enTypeOfBacNetFunktion.Type_Zähler,		enTypeOfBacNetTextListIn := enTypeOfBacNetTextList.EVENTMESSAGE	),	'B_TL_1_ToNormal'		));		

		(* Ziel												Convert			BacNet Text		Textlistname									BacNet Funktion																BacNet Textlist type												TextId		*)	
		B_TL_1.udiNotificationClass						:= 	TO_UDINT	(	fcGetBcText(	GVL_BACNET.fbBacNetParameter.metGetTextListName(enTypeOfBacNetFunktionIn := enTypeOfBacNetFunktion.Type_Zähler,		enTypeOfBacNetTextListIn := enTypeOfBacNetTextList.NC		),	'B_TL_1_NC'	));	
		B_TL_1.eNotifyType								:= 	WagoTypesBACnet.eBACnetNotifyType.NOTIFY_TYPE_EVENT;

		(* Logging Type *)
		B_TL_1.eLoggingType								:= WagoTypesBACnet.eBACnetLoggingType.LOGGING_TYPE_POLLED;
		
		(* Activate Logging *)
		B_TL_1.xEnable	:= TRUE;
	ELSE
		B_TL_1.Delete();
	END_IF;
	(* Get Status *)
	metCreate_B_TL_1 := B_TL_1.xIsCreated;	
END_IF;
END_METHOD

METHOD metCreate_C_BV_1 : BOOL
(* C_BV_1*)
IF NOT C_BV_1.xIsCreated THEN
	(* Ziel						UTF8->ASCII						OBJ_NAME_BASE			BacNet Text		Textlistname									BacNet Funktion																BacNet Textlist type												TextId		*)
	C_BV_1._sObjectName		:=	fcUtfToAscii(Standard.CONCAT(	OBJ_NAME_BASE		,	fcGetBcText(	GVL_BACNET.fbBacNetParameter.metGetTextListName(enTypeOfBacNetFunktionIn := enTypeOfBacNetFunktion.Type_Zähler,		enTypeOfBacNetTextListIn := enTypeOfBacNetTextList.ENDING		),	'C_BV_1')));
	C_BV_1._sDescription	:= 	fcUtfToAscii(Standard.CONCAT(	OBJ_NAME_DESCRIPTION,	fcGetBcText(	GVL_BACNET.fbBacNetParameter.metGetTextListName(enTypeOfBacNetFunktionIn := enTypeOfBacNetFunktion.Type_Zähler,		enTypeOfBacNetTextListIn := enTypeOfBacNetTextList.DESCRIPTION	),	'C_BV_1')));
	(* Create Id from Base Id and Object Nr (Last nummber of Name *)	
	C_BV_1.Create(diInstance := TO_DINT(Standard.CONCAT(TO_STRING(dwOBJ_ID_BASE),'1')));
	(* Check if Created *)
	IF C_BV_1.xIsCreated THEN
		(* Set Group *)
		C_BV_1.setPropertyGroup(WagoTypesBacNet.eBACnetPropertyIdentifier.PROP_PRESENT_VALUE						,WagoTypesBacNet.eBACnetPropertyUpdateGroup.GROUP_CYCLIC);
		C_BV_1.setPropertyGroup(WagoTypesBacNet.eBACnetPropertyIdentifier.PROP_PRIORITY_ARRAY						,WagoTypesBacNet.eBACnetPropertyUpdateGroup.GROUP_CYCLIC);
		C_BV_1.setPropertyGroup(WagoTypesBacNet.eBACnetPropertyIdentifier.PROP_ELAPSED_ACTIVE_TIME					,WagoTypesBacNet.eBACnetPropertyUpdateGroup.GROUP_CYCLIC);
		C_BV_1.setPropertyGroup(WagoTypesBacNet.eBACnetPropertyIdentifier.PROP_DESCRIPTION							,WagoTypesBacNet.eBACnetPropertyUpdateGroup.GROUP_CYCLIC);
		C_BV_1.setPropertyGroup(WagoTypesBacNet.eBACnetPropertyIdentifier.PROP_EVENT_MESSAGE_TEXTS_CONFIG			,WagoTypesBacNet.eBACnetPropertyUpdateGroup.GROUP_CYCLIC);
		(* Set Description to Overwrite retain*)
		C_BV_1.sDescription	:= C_BV_1._sDescription;
		(* Ziel												UTF8->ASCII		BacNet Text		Textlistname									BacNet Funktion																BacNet Textlist type												TextId		*)
		C_BV_1.IEventMessageTextsConfig.sToOffNormal	:=	fcUtfToAscii(	fcGetBcText(	GVL_BACNET.fbBacNetParameter.metGetTextListName(enTypeOfBacNetFunktionIn := enTypeOfBacNetFunktion.Type_Zähler,		enTypeOfBacNetTextListIn := enTypeOfBacNetTextList.EVENTMESSAGE	),	'C_BV_1_ToOffNormal'	));		
		C_BV_1.IEventMessageTextsConfig.sToFault		:=	fcUtfToAscii(	fcGetBcText(	GVL_BACNET.fbBacNetParameter.metGetTextListName(enTypeOfBacNetFunktionIn := enTypeOfBacNetFunktion.Type_Zähler,		enTypeOfBacNetTextListIn := enTypeOfBacNetTextList.EVENTMESSAGE	),	'C_BV_1_ToFault'		));		
		C_BV_1.IEventMessageTextsConfig.sToNormal		:=	fcUtfToAscii(	fcGetBcText(	GVL_BACNET.fbBacNetParameter.metGetTextListName(enTypeOfBacNetFunktionIn := enTypeOfBacNetFunktion.Type_Zähler,		enTypeOfBacNetTextListIn := enTypeOfBacNetTextList.EVENTMESSAGE	),	'C_BV_1_ToNormal'		));		

		(* Ziel												UTF8->ASCII		BacNet Text		Textlistname									BacNet Funktion																BacNet Textlist type												TextId		*)	
		C_BV_1.sActiveText								:= 	fcUtfToAscii(	fcGetBcText(	GVL_BACNET.fbBacNetParameter.metGetTextListName(enTypeOfBacNetFunktionIn := enTypeOfBacNetFunktion.Type_Zähler,		enTypeOfBacNetTextListIn := enTypeOfBacNetTextList.PRESENTVALUE	),	'C_BV_1_ST_ACTIVE'		));
		C_BV_1.sInactiveText							:= 	fcUtfToAscii(	fcGetBcText(	GVL_BACNET.fbBacNetParameter.metGetTextListName(enTypeOfBacNetFunktionIn := enTypeOfBacNetFunktion.Type_Zähler,		enTypeOfBacNetTextListIn := enTypeOfBacNetTextList.PRESENTVALUE	),	'C_BV_1_ST_INACTIVE'	));	

		(* Ziel												Convert			BacNet Text		Textlistname									BacNet Funktion																	BacNet Textlist type											TextId		*)	
		C_BV_1.udiNotificationClass						:= 	TO_UDINT	(	fcGetBcText(	GVL_BACNET.fbBacNetParameter.metGetTextListName(enTypeOfBacNetFunktionIn := enTypeOfBacNetFunktion.Type_Zähler,		enTypeOfBacNetTextListIn := enTypeOfBacNetTextList.NC			),	'C_BV_1_NC'	));	
		C_BV_1.eNotifyType								:= 	WagoTypesBACnet.eBACnetNotifyType.NOTIFY_TYPE_ALARM;		
		C_BV_1.xAlarmValue								:= 	TO_BOOL		(	fcGetBcText(	GVL_BACNET.fbBacNetParameter.metGetTextListName(enTypeOfBacNetFunktionIn := enTypeOfBacNetFunktion.Type_Zähler,		enTypeOfBacNetTextListIn := enTypeOfBacNetTextList.NC			),	'C_BV_1_ALV'	));	
		
	ELSE
		C_BV_1.Delete();
	END_IF;
	(* Get Status *)
	metCreate_C_BV_1 := C_BV_1.xIsCreated;	
END_IF;
END_METHOD

METHOD metCREATE : BOOL;
VAR_INPUT
END_VAR
VAR
	usiErrors	:	USINT;
END_VAR
(* Get Revision *)
CASE GVL_BACNET.fbBacNetParameter.proKBOB_REV OF
	(* KBOB 2021 V2 *)
	enKBOB_REV.KBOB_REV2021_V2:
		usiErrors := usiErrors + TO_USINT(NOT metCREATE_KBOB_2021_V2());
	(* KBOB 2017 V1 *)
	enKBOB_REV.KBOB_REV2017_V1:
		usiErrors := usiErrors + TO_USINT(NOT metCREATE_KBOB_2017_V1());
	(* Default *)
	ELSE
		usiErrors := usiErrors + TO_USINT(NOT metCREATE_KBOB_2021_V2());
END_CASE;

(* OK = 0*)
xErrorCreate := TO_BOOL(usiErrors);
metCREATE := NOT TO_BOOL(usiErrors) AND usiCreateCase = usiAnzBacNetObj;
END_METHOD

METHOD metCREATE_KBOB_2017_V1 : BOOL;
VAR_INPUT
END_VAR
VAR
	oStatus		:	WagoSysErrorBase.FbResult;
END_VAR
(* Resett *)
usiErrors := 0;	

(* Create Objeccts *)
CASE usiCreateCase OF
	1:	
		usiErrors := usiErrors + TO_USINT(NOT metCreate_A_AV_1());
	2:
		usiErrors := usiErrors + TO_USINT(NOT metCreate_B_TL_1());
	3:	
		usiErrors := usiErrors + TO_USINT(NOT metCreate_C_BV_1());
	0: 
		usiCreateCase := 1;
ELSE
	usiCreateCase := 0;
END_CASE;

(* STRUCT VIEW *)
metCREATE_STRUCTVIEW_KBOB_2017_V1();

(* OK = 0*)
metCREATE_KBOB_2017_V1 := NOT TO_BOOL(usiErrors);
END_METHOD

METHOD metCREATE_STRUCTVIEW_KBOB_2017_V1 : BOOL
VAR_INPUT
END_VAR
CASE usiCreateCase OF
	1:	
		fcXMLStructuredView(THIS^,A_AV_1.IObjectIdentifier);
	2:
		fcXMLStructuredView(THIS^,B_TL_1.IObjectIdentifier);
	3:
		fcXMLStructuredView(THIS^,C_BV_1.IObjectIdentifier);
		fcXMLAddStructuredViewToDevice(THIS^);
	0: 
		usiCreateCase := 1;
ELSE
	usiCreateCase := 0;
END_CASE
END_METHOD

METHOD metDELETE : BOOL
VAR_INPUT
END_VAR
VAR
	oStatus		:	WagoSysErrorBase.FbResult;
	usiErrors	:	USINT;
END_VAR
(* A_AV_1*)
IF A_AV_1.xIsCreated THEN
	A_AV_1.Delete(oStatus=>oStatus);	
END_IF;
(* B_TL_1 *)
IF B_TL_1.xIsCreated THEN
	IF GVL_BACNET.fbBacNetParameter.proDestroyBacNetOverrideXmlNode THEN
		fcXMLDeleteOverrideNode(fcBacNetIdToIdWitType(B_TL_1.IObjectIdentifier.diInstance,B_TL_1.IObjectIdentifier.eObjectType));
	END_IF;
	B_TL_1.Delete(oStatus=>oStatus);
END_IF;
(* C_BV_1 *)
IF C_BV_1.xIsCreated THEN
	C_BV_1.Delete(oStatus=>oStatus);
END_IF;
(* Delete Struct View *)
IF GVL_BACNET.fbBacNetParameter.proDestroyBacNetOverrideXmlNode THEN
	fcXMLDeleteOverrideNode(fcBacNetIdToIdWitType(TO_DINT(CONCAT(TO_STRING(OBJ_ID_BASE),'1')),WagoTypesBacNet.eBACnetObjectType.BACnet_structured_view));
	fcXMLDeleteStructuredViewFromDevice(fcBacNetIdToIdWitType(TO_DINT(CONCAT(TO_STRING(OBJ_ID_BASE),'1')),WagoTypesBacNet.eBACnetObjectType.BACnet_structured_view));
END_IF;
metDELETE :=	A_AV_1.xIsCreated OR
				B_TL_1.xIsCreated OR
				C_BV_1.xIsCreated;
(* Reset Create Case *)
usiCreateCase := 1;
END_METHOD

(*FB_Exit muss explizit implementiert werden. Wenn es eine Implementierung gibt, dann wird 
die Methode aufgerufen, bevor die Steuerung den Code der Funktionsbaustein-Instanz entfernt
(impliziter Aufruf. Der Rückgabewert wird nicht ausgewertet.*)
METHOD FB_Exit : BOOL
VAR_INPUT
	(* TRUE: Die Exit-Methode wird aufgerufen, um die Instanz zu verlassen, die hinterher kopiert wird Online-Change).  *)
	bInCopyCode	: BOOL;
END_VAR
(* A_AV_1*)
IF A_AV_1.xIsCreated THEN
	A_AV_1.Delete();	
END_IF;
(* B_TL_1 *)
IF B_TL_1.xIsCreated THEN
	B_TL_1.Delete();
END_IF;
(* C_BV_1 *)
IF C_BV_1.xIsCreated THEN
	C_BV_1.Delete();
END_IF;
END_METHOD

METHOD metCYCLIC_DESCRIPTION_FIX
VAR_INPUT
END_VAR
(* A_AV_1 *)
IF A_AV_1.xIsCreated THEN
	IF A_AV_1.sDescription <> A_AV_1._sDescription THEN
		A_AV_1.sDescription := A_AV_1._sDescription;
	END_IF;
END_IF;

(* B_TL_1 *)
IF B_TL_1.xIsCreated THEN
	IF B_TL_1.sDescription <> B_TL_1._sDescription THEN
		B_TL_1.sDescription := B_TL_1._sDescription;
	END_IF;
END_IF;

(* C_BV_1 *)
IF C_BV_1.xIsCreated THEN
	IF C_BV_1.sDescription <> C_BV_1._sDescription THEN
		C_BV_1.sDescription := C_BV_1._sDescription;
	END_IF;
END_IF;
END_METHOD

METHOD metCYCLIC_KBOB_2017_V1
VAR_INPUT
END_VAR
(* A_BI_1 *)
IF A_AV_1.rPresentValue <> rValue THEN
	A_AV_1.rPresentValue := rValue;				
END_IF;	
(* C_BV_1 *)
IF C_BV_1.xPresentValue <> xError THEN
	C_BV_1.xPresentValue := xError;				
END_IF;
END_METHOD

METHOD metCYCLIC_KBOB_2021_V2
VAR_INPUT
END_VAR
(* A_BI_1 *)
IF A_AV_1.rPresentValue <> rValue THEN
	A_AV_1.rPresentValue := rValue;				
END_IF;	
(* C_BV_1 *)
IF C_BV_1.xPresentValue <> xError THEN
	C_BV_1.xPresentValue := xError;				
END_IF;
END_METHOD

END_FUNCTION_BLOCK

// 30 Program Organization Units/FBs/AT_FUNKTIONEN/AT_STELLORGAN_STETIG/FB_AT_AT_STELLORGAN_STETIG
FUNCTION_BLOCK FB_AT_AT_STELLORGAN_STETIG EXTENDS FB_OBJ_ID_BASE
VAR_INPUT
	xRelease			:	BOOL;
	rRelease			:	REAL;
	xSafetyOk			:	BOOL;		
	xHand				:	BOOL;
	rAcknowledge		:	REAL;
	xAcknowledgeZu		:	BOOL;
	xAcknowledgeAuf		:	BOOL;
	xErrorStellorgan	:	BOOL;
END_VAR
VAR_OUTPUT
	(* Requests *)
	xHandPrio8			:	BOOL;
	rDemandeHandPrio8	:	REAL;
END_VAR
VAR
	(* BacNet Objects *)
	A_AO_1				:	WagoSysBACnet.FbAnalogOutput_large(-1);					// Stellwert
	B_AI_1				:	WagoSysBACnet.FbAnalogInput_large(-1);					// Istwert
	C_TL_1				:	WagoSysBACnet.FbTrendLog_large(-1);                     // Aufzeichnung Stellwert
	D_BI_1				:	WagoSysBACnet.FbBinaryInput_large(-1);					// Stellungsrückmeldung ZU
	E_BI_2				:	WagoSysBACnet.FbBinaryInput_large(-1);					// Stellungsrückmeldung AUF
	F_BV_1				:	WagoSysBACnet.FbBinaryValue_large(-1);					// Störung Stellorgan
END_VAR
VAR CONSTANT
	usiAnzBacNetObj	:	USINT	:= 6;
END_VAR

(* Call Base FB*)
SUPER^();
(* Cyclic Action *)
IF xCreatet THEN
	(* DESCTIPTION FIX *)
	metCYCLIC_DESCRIPTION_FIX();
	(* Get Revision *)
	CASE GVL_BACNET.fbBacNetParameter.proKBOB_REV OF
		(* KBOB 2021 V2 *)
		enKBOB_REV.KBOB_REV2021_V2:
			metCYCLIC_KBOB_2021_V2();
		(* KBOB 2017 V1 *)
		enKBOB_REV.KBOB_REV2017_V1:
			metCYCLIC_KBOB_2017_V1();
		(* Default *)
		ELSE
			metCYCLIC_KBOB_2021_V2();
	END_CASE;	
END_IF;

METHOD metCREATE_STRUCTVIEW_KBOB_2021_V2 : BOOL
VAR_INPUT
END_VAR
CASE usiCreateCase OF
	1:
		fcXMLStructuredView(THIS^,A_AO_1.IObjectIdentifier);
	2:
		fcXMLStructuredView(THIS^,B_AI_1.IObjectIdentifier);
	3:
		fcXMLStructuredView(THIS^,C_TL_1.IObjectIdentifier);
	4:
		fcXMLStructuredView(THIS^,D_BI_1.IObjectIdentifier);
	5:
		fcXMLStructuredView(THIS^,E_BI_2.IObjectIdentifier);
	6:
		fcXMLStructuredView(THIS^,F_BV_1.IObjectIdentifier);
		fcXMLAddStructuredViewToDevice(THIS^);	
	0: 
		usiCreateCase := 1;
ELSE
	usiCreateCase := 0;
END_CASE
END_METHOD

METHOD metCREATE_KBOB_2021_V2 : BOOL;
VAR_INPUT
END_VAR
VAR
	oStatus		:	WagoSysErrorBase.FbResult;
	usiErrors	:	USINT;
END_VAR
(* Resett *)
usiErrors := 0;	

(* Create Objeccts *)
CASE usiCreateCase OF
	1:	
		usiErrors := usiErrors + TO_USINT(NOT metCreate_A_AO_1());
	2:
		usiErrors := usiErrors + TO_USINT(NOT metCreate_B_AI_1());
	3:	
		usiErrors := usiErrors + TO_USINT(NOT metCreate_C_TL_1());
	4:	
		usiErrors := usiErrors + TO_USINT(NOT metCreate_D_BI_1());
	5:
		usiErrors := usiErrors + TO_USINT(NOT metCreate_E_BI_2());
	6:	
		usiErrors := usiErrors + TO_USINT(NOT metCreate_F_BV_1());
	0: 
		usiCreateCase := 1;
ELSE
	usiCreateCase := 0;
END_CASE;

(* STRUCT VIEW *)
metCREATE_STRUCTVIEW_KBOB_2021_V2();

(* OK = 0*)
metCREATE_KBOB_2021_V2 := NOT TO_BOOL(usiErrors);
END_METHOD

METHOD metCreate_D_BI_1 : BOOL
(* D_BI_1*)
IF NOT D_BI_1.xIsCreated THEN
	(* Ziel						UTF8->ASCII						OBJ_NAME_BASE			BacNet Text		Textlistname									BacNet Funktion																BacNet Textlist type												TextId		*)
	D_BI_1._sObjectName		:=	fcUtfToAscii(Standard.CONCAT(	OBJ_NAME_BASE		,	fcGetBcText(	GVL_BACNET.fbBacNetParameter.metGetTextListName(enTypeOfBacNetFunktionIn := enTypeOfBacNetFunktion.Type_AntriebStetig,		enTypeOfBacNetTextListIn := enTypeOfBacNetTextList.ENDING		),	'D_BI_1')));
	D_BI_1._sDescription	:= 	fcUtfToAscii(Standard.CONCAT(	OBJ_NAME_DESCRIPTION,	fcGetBcText(	GVL_BACNET.fbBacNetParameter.metGetTextListName(enTypeOfBacNetFunktionIn := enTypeOfBacNetFunktion.Type_AntriebStetig,		enTypeOfBacNetTextListIn := enTypeOfBacNetTextList.DESCRIPTION	),	'D_BI_1')));
	(* Create Id from Base Id and Object Nr (Last nummber of Name *)	
	D_BI_1.Create(diInstance := TO_DINT(Standard.CONCAT(TO_STRING(dwOBJ_ID_BASE),'1')));
	(* Check if Created *)
	IF D_BI_1.xIsCreated THEN
		(* Set Group *)
		D_BI_1.setPropertyGroup(WagoTypesBacNet.eBACnetPropertyIdentifier.PROP_PRESENT_VALUE						,WagoTypesBacNet.eBACnetPropertyUpdateGroup.GROUP_CYCLIC);
		D_BI_1.setPropertyGroup(WagoTypesBacNet.eBACnetPropertyIdentifier.PROP_PRIORITY_ARRAY						,WagoTypesBacNet.eBACnetPropertyUpdateGroup.GROUP_CYCLIC);
		D_BI_1.setPropertyGroup(WagoTypesBacNet.eBACnetPropertyIdentifier.PROP_ELAPSED_ACTIVE_TIME					,WagoTypesBacNet.eBACnetPropertyUpdateGroup.GROUP_CYCLIC);
		D_BI_1.setPropertyGroup(WagoTypesBacNet.eBACnetPropertyIdentifier.PROP_DESCRIPTION							,WagoTypesBacNet.eBACnetPropertyUpdateGroup.GROUP_CYCLIC);
		D_BI_1.setPropertyGroup(WagoTypesBacNet.eBACnetPropertyIdentifier.PROP_EVENT_MESSAGE_TEXTS_CONFIG			,WagoTypesBacNet.eBACnetPropertyUpdateGroup.GROUP_CYCLIC);
				
		(* Ziel												UTF8->ASCII		BacNet Text		Textlistname									BacNet Funktion																BacNet Textlist type												TextId		*)
		D_BI_1.IEventMessageTextsConfig.sToOffNormal	:=	fcUtfToAscii(	fcGetBcText(	GVL_BACNET.fbBacNetParameter.metGetTextListName(enTypeOfBacNetFunktionIn := enTypeOfBacNetFunktion.Type_AntriebStetig,		enTypeOfBacNetTextListIn := enTypeOfBacNetTextList.EVENTMESSAGE	),	'D_BI_1_ToOffNormal'	));		
		D_BI_1.IEventMessageTextsConfig.sToFault		:=	fcUtfToAscii(	fcGetBcText(	GVL_BACNET.fbBacNetParameter.metGetTextListName(enTypeOfBacNetFunktionIn := enTypeOfBacNetFunktion.Type_AntriebStetig,		enTypeOfBacNetTextListIn := enTypeOfBacNetTextList.EVENTMESSAGE	),	'D_BI_1_ToFault'		));		
		D_BI_1.IEventMessageTextsConfig.sToNormal		:=	fcUtfToAscii(	fcGetBcText(	GVL_BACNET.fbBacNetParameter.metGetTextListName(enTypeOfBacNetFunktionIn := enTypeOfBacNetFunktion.Type_AntriebStetig,		enTypeOfBacNetTextListIn := enTypeOfBacNetTextList.EVENTMESSAGE	),	'D_BI_1_ToNormal'		));		

		(* Ziel												UTF8->ASCII		BacNet Text		Textlistname									BacNet Funktion																BacNet Textlist type												TextId		*)	
		D_BI_1.sActiveText								:= 	fcUtfToAscii(	fcGetBcText(	GVL_BACNET.fbBacNetParameter.metGetTextListName(enTypeOfBacNetFunktionIn := enTypeOfBacNetFunktion.Type_AntriebStetig,		enTypeOfBacNetTextListIn := enTypeOfBacNetTextList.PRESENTVALUE	),	'D_BI_1_ST_ACTIVE'		));
		D_BI_1.sInactiveText							:= 	fcUtfToAscii(	fcGetBcText(	GVL_BACNET.fbBacNetParameter.metGetTextListName(enTypeOfBacNetFunktionIn := enTypeOfBacNetFunktion.Type_AntriebStetig,		enTypeOfBacNetTextListIn := enTypeOfBacNetTextList.PRESENTVALUE	),	'D_BI_1_ST_INACTIVE'	));	

		(* Ziel												Convert			BacNet Text		Textlistname									BacNet Funktion																BacNet Textlist type												TextId		*)	
		D_BI_1.udiNotificationClass						:= 	TO_UDINT	(	fcGetBcText(	GVL_BACNET.fbBacNetParameter.metGetTextListName(enTypeOfBacNetFunktionIn := enTypeOfBacNetFunktion.Type_AntriebStetig,		enTypeOfBacNetTextListIn := enTypeOfBacNetTextList.NC			),	'D_BI_1_NC'	));	
		D_BI_1.eNotifyType								:= 	WagoTypesBACnet.eBACnetNotifyType.NOTIFY_TYPE_EVENT;
		D_BI_1.xAlarmValue								:= 	TO_BOOL		(	fcGetBcText(	GVL_BACNET.fbBacNetParameter.metGetTextListName(enTypeOfBacNetFunktionIn := enTypeOfBacNetFunktion.Type_AntriebStetig,		enTypeOfBacNetTextListIn := enTypeOfBacNetTextList.NC			),	'D_BI_1_ALV'	));	
		
	ELSE
		D_BI_1.Delete();
	END_IF;
	(* Get Status *)
	metCreate_D_BI_1 := D_BI_1.xIsCreated;	
END_IF;
END_METHOD

METHOD metCreate_A_AO_1 : BOOL
(* A_AO_1*)
IF NOT A_AO_1.xIsCreated THEN
	(* Ziel						UTF8->ASCII						OBJ_NAME_BASE			BacNet Text		Textlistname									BacNet Funktion																BacNet Textlist type												TextId		*)
	A_AO_1._sObjectName		:=	fcUtfToAscii(Standard.CONCAT(	OBJ_NAME_BASE		,	fcGetBcText(	GVL_BACNET.fbBacNetParameter.metGetTextListName(enTypeOfBacNetFunktionIn := enTypeOfBacNetFunktion.Type_AntriebStetig,		enTypeOfBacNetTextListIn := enTypeOfBacNetTextList.ENDING		),	'A_AO_1')));
	A_AO_1._sDescription	:= 	fcUtfToAscii(Standard.CONCAT(	OBJ_NAME_DESCRIPTION,	fcGetBcText(	GVL_BACNET.fbBacNetParameter.metGetTextListName(enTypeOfBacNetFunktionIn := enTypeOfBacNetFunktion.Type_AntriebStetig,		enTypeOfBacNetTextListIn := enTypeOfBacNetTextList.DESCRIPTION	),	'A_AO_1')));
	(* Create Id from Base Id and Object Nr (Last nummber of Name *)	
	A_AO_1.Create(diInstance := TO_DINT(Standard.CONCAT(TO_STRING(dwOBJ_ID_BASE),'1')));
	(* Check if Created *)
	IF A_AO_1.xIsCreated THEN
		(* Set Group *)
		A_AO_1.setPropertyGroup(WagoTypesBacNet.eBACnetPropertyIdentifier.PROP_PRESENT_VALUE						,WagoTypesBacNet.eBACnetPropertyUpdateGroup.GROUP_CYCLIC);
		A_AO_1.setPropertyGroup(WagoTypesBacNet.eBACnetPropertyIdentifier.PROP_PRIORITY_ARRAY						,WagoTypesBacNet.eBACnetPropertyUpdateGroup.GROUP_CYCLIC);
		A_AO_1.setPropertyGroup(WagoTypesBacNet.eBACnetPropertyIdentifier.PROP_ELAPSED_ACTIVE_TIME					,WagoTypesBacNet.eBACnetPropertyUpdateGroup.GROUP_CYCLIC);
		A_AO_1.setPropertyGroup(WagoTypesBacNet.eBACnetPropertyIdentifier.PROP_DESCRIPTION							,WagoTypesBacNet.eBACnetPropertyUpdateGroup.GROUP_CYCLIC);
		A_AO_1.setPropertyGroup(WagoTypesBacNet.eBACnetPropertyIdentifier.PROP_EVENT_MESSAGE_TEXTS_CONFIG			,WagoTypesBacNet.eBACnetPropertyUpdateGroup.GROUP_CYCLIC);
			
		(* Ziel												UTF8->ASCII		BacNet Text		Textlistname									BacNet Funktion																BacNet Textlist type												TextId		*)
		A_AO_1.IEventMessageTextsConfig.sToOffNormal	:=	fcUtfToAscii(	fcGetBcText(	GVL_BACNET.fbBacNetParameter.metGetTextListName(enTypeOfBacNetFunktionIn := enTypeOfBacNetFunktion.Type_AntriebStetig,		enTypeOfBacNetTextListIn := enTypeOfBacNetTextList.EVENTMESSAGE	),	'A_AO_1_ToOffNormal'	));		
		A_AO_1.IEventMessageTextsConfig.sToFault		:=	fcUtfToAscii(	fcGetBcText(	GVL_BACNET.fbBacNetParameter.metGetTextListName(enTypeOfBacNetFunktionIn := enTypeOfBacNetFunktion.Type_AntriebStetig,		enTypeOfBacNetTextListIn := enTypeOfBacNetTextList.EVENTMESSAGE	),	'A_AO_1_ToFault'		));		
		A_AO_1.IEventMessageTextsConfig.sToNormal		:=	fcUtfToAscii(	fcGetBcText(	GVL_BACNET.fbBacNetParameter.metGetTextListName(enTypeOfBacNetFunktionIn := enTypeOfBacNetFunktion.Type_AntriebStetig,		enTypeOfBacNetTextListIn := enTypeOfBacNetTextList.EVENTMESSAGE	),	'A_AO_1_ToNormal'		));		


		(* Ziel												Convert			BacNet Text		Textlistname									BacNet Funktion																BacNet Textlist type												TextId		*)	
		A_AO_1.udiNotificationClass						:= 	TO_UDINT	(	fcGetBcText(	GVL_BACNET.fbBacNetParameter.metGetTextListName(enTypeOfBacNetFunktionIn := enTypeOfBacNetFunktion.Type_AntriebStetig,		enTypeOfBacNetTextListIn := enTypeOfBacNetTextList.NC			),	'A_AO_1_NC'	));	
		A_AO_1.eNotifyType								:= 	WagoTypesBACnet.eBACnetNotifyType.NOTIFY_TYPE_EVENT;
		
	ELSE
		A_AO_1.Delete();
	END_IF;
	(* Get Status *)
	metCreate_A_AO_1 := A_AO_1.xIsCreated;	
END_IF;
END_METHOD

METHOD metCreate_C_TL_1 : BOOL
VAR

END_VAR
(* C_TL_1*)
IF NOT C_TL_1.xIsCreated THEN
	(* Ziel						UTF8->ASCII						OBJ_NAME_BASE			BacNet Text		Textlistname									BacNet Funktion																BacNet Textlist type												TextId		*)
	C_TL_1._sObjectName		:=	fcUtfToAscii(Standard.CONCAT(	OBJ_NAME_BASE		,	fcGetBcText(	GVL_BACNET.fbBacNetParameter.metGetTextListName(enTypeOfBacNetFunktionIn := enTypeOfBacNetFunktion.Type_AntriebStetig,		enTypeOfBacNetTextListIn := enTypeOfBacNetTextList.ENDING		),	'C_TL_1')));
	C_TL_1._sDescription	:= 	fcUtfToAscii(Standard.CONCAT(	OBJ_NAME_DESCRIPTION,	fcGetBcText(	GVL_BACNET.fbBacNetParameter.metGetTextListName(enTypeOfBacNetFunktionIn := enTypeOfBacNetFunktion.Type_AntriebStetig,		enTypeOfBacNetTextListIn := enTypeOfBacNetTextList.DESCRIPTION	),	'C_TL_1')));
	(* Create Id from Base Id and Object Nr (Last nummber of Name *)	
	C_TL_1.Create(diInstance := TO_DINT(Standard.CONCAT(TO_STRING(dwOBJ_ID_BASE),'1')));
	(* Check if Created *)
	IF C_TL_1.xIsCreated THEN
		(* Set Group *)
		C_TL_1.setPropertyGroup(WagoTypesBacNet.eBACnetPropertyIdentifier.PROP_PRESENT_VALUE						,WagoTypesBacNet.eBACnetPropertyUpdateGroup.GROUP_CYCLIC);
		C_TL_1.setPropertyGroup(WagoTypesBacNet.eBACnetPropertyIdentifier.PROP_PRIORITY_ARRAY						,WagoTypesBacNet.eBACnetPropertyUpdateGroup.GROUP_CYCLIC);
		C_TL_1.setPropertyGroup(WagoTypesBacNet.eBACnetPropertyIdentifier.PROP_ELAPSED_ACTIVE_TIME					,WagoTypesBacNet.eBACnetPropertyUpdateGroup.GROUP_CYCLIC);
		C_TL_1.setPropertyGroup(WagoTypesBacNet.eBACnetPropertyIdentifier.PROP_DESCRIPTION							,WagoTypesBacNet.eBACnetPropertyUpdateGroup.GROUP_CYCLIC);
		C_TL_1.setPropertyGroup(WagoTypesBacNet.eBACnetPropertyIdentifier.PROP_EVENT_MESSAGE_TEXTS_CONFIG			,WagoTypesBacNet.eBACnetPropertyUpdateGroup.GROUP_CYCLIC);
		
		(* Crate Override *)
		fcXMLTrendLogOverride(C_TL_1,A_AO_1.IObjectIdentifier,WagoTypesBacNet.eBACnetPropertyIdentifier.PROP_FEEDBACK_VALUE);
		
		(* Ziel												UTF8->ASCII		BacNet Text		Textlistname									BacNet Funktion																BacNet Textlist type												TextId		*)
		C_TL_1.IEventMessageTextsConfig.sToOffNormal	:=	fcUtfToAscii(	fcGetBcText(	GVL_BACNET.fbBacNetParameter.metGetTextListName(enTypeOfBacNetFunktionIn := enTypeOfBacNetFunktion.Type_AntriebStetig,		enTypeOfBacNetTextListIn := enTypeOfBacNetTextList.EVENTMESSAGE	),	'C_TL_1_ToOffNormal'	));		
		C_TL_1.IEventMessageTextsConfig.sToFault		:=	fcUtfToAscii(	fcGetBcText(	GVL_BACNET.fbBacNetParameter.metGetTextListName(enTypeOfBacNetFunktionIn := enTypeOfBacNetFunktion.Type_AntriebStetig,		enTypeOfBacNetTextListIn := enTypeOfBacNetTextList.EVENTMESSAGE	),	'C_TL_1_ToFault'		));		
		C_TL_1.IEventMessageTextsConfig.sToNormal		:=	fcUtfToAscii(	fcGetBcText(	GVL_BACNET.fbBacNetParameter.metGetTextListName(enTypeOfBacNetFunktionIn := enTypeOfBacNetFunktion.Type_AntriebStetig,		enTypeOfBacNetTextListIn := enTypeOfBacNetTextList.EVENTMESSAGE	),	'C_TL_1_ToNormal'		));		

		(* Ziel												Convert			BacNet Text		Textlistname									BacNet Funktion																BacNet Textlist type												TextId		*)	
		C_TL_1.udiNotificationClass						:= 	TO_UDINT	(	fcGetBcText(	GVL_BACNET.fbBacNetParameter.metGetTextListName(enTypeOfBacNetFunktionIn := enTypeOfBacNetFunktion.Type_AntriebStetig,		enTypeOfBacNetTextListIn := enTypeOfBacNetTextList.NC		),	'C_TL_1_NC'	));	
		C_TL_1.eNotifyType								:= 	WagoTypesBACnet.eBACnetNotifyType.NOTIFY_TYPE_EVENT;
		
		(* Logging Type *)
		C_TL_1.eLoggingType								:= WagoTypesBACnet.eBACnetLoggingType.LOGGING_TYPE_POLLED;
		
		(* Activate Logging *)
		C_TL_1.xEnable	:= TRUE;	
								
	ELSE
		C_TL_1.Delete();
	END_IF;
	(* Get Status *)
	metCreate_C_TL_1 := C_TL_1.xIsCreated;	
END_IF;
END_METHOD

METHOD metCreate_E_BI_2 : BOOL
(* E_BI_2*)
IF NOT E_BI_2.xIsCreated THEN
	(* Ziel						UTF8->ASCII						OBJ_NAME_BASE			BacNet Text		Textlistname									BacNet Funktion																BacNet Textlist type												TextId		*)
	E_BI_2._sObjectName		:=	fcUtfToAscii(Standard.CONCAT(	OBJ_NAME_BASE		,	fcGetBcText(	GVL_BACNET.fbBacNetParameter.metGetTextListName(enTypeOfBacNetFunktionIn := enTypeOfBacNetFunktion.Type_AntriebStetig,		enTypeOfBacNetTextListIn := enTypeOfBacNetTextList.ENDING		),	'E_BI_2')));
	E_BI_2._sDescription	:= 	fcUtfToAscii(Standard.CONCAT(	OBJ_NAME_DESCRIPTION,	fcGetBcText(	GVL_BACNET.fbBacNetParameter.metGetTextListName(enTypeOfBacNetFunktionIn := enTypeOfBacNetFunktion.Type_AntriebStetig,		enTypeOfBacNetTextListIn := enTypeOfBacNetTextList.DESCRIPTION	),	'E_BI_2')));
	(* Create Id from Base Id and Object Nr (Last nummber of Name *)	
	E_BI_2.Create(diInstance := TO_DINT(Standard.CONCAT(TO_STRING(dwOBJ_ID_BASE),'2')));
	(* Check if Created *)
	IF E_BI_2.xIsCreated THEN
		(* Set Group *)
		E_BI_2.setPropertyGroup(WagoTypesBacNet.eBACnetPropertyIdentifier.PROP_PRESENT_VALUE						,WagoTypesBacNet.eBACnetPropertyUpdateGroup.GROUP_CYCLIC);
		E_BI_2.setPropertyGroup(WagoTypesBacNet.eBACnetPropertyIdentifier.PROP_PRIORITY_ARRAY						,WagoTypesBacNet.eBACnetPropertyUpdateGroup.GROUP_CYCLIC);
		E_BI_2.setPropertyGroup(WagoTypesBacNet.eBACnetPropertyIdentifier.PROP_ELAPSED_ACTIVE_TIME					,WagoTypesBacNet.eBACnetPropertyUpdateGroup.GROUP_CYCLIC);
		E_BI_2.setPropertyGroup(WagoTypesBacNet.eBACnetPropertyIdentifier.PROP_DESCRIPTION							,WagoTypesBacNet.eBACnetPropertyUpdateGroup.GROUP_CYCLIC);
		E_BI_2.setPropertyGroup(WagoTypesBacNet.eBACnetPropertyIdentifier.PROP_EVENT_MESSAGE_TEXTS_CONFIG			,WagoTypesBacNet.eBACnetPropertyUpdateGroup.GROUP_CYCLIC);
				
		(* Ziel												UTF8->ASCII		BacNet Text		Textlistname									BacNet Funktion																BacNet Textlist type												TextId		*)
		E_BI_2.IEventMessageTextsConfig.sToOffNormal	:=	fcUtfToAscii(	fcGetBcText(	GVL_BACNET.fbBacNetParameter.metGetTextListName(enTypeOfBacNetFunktionIn := enTypeOfBacNetFunktion.Type_AntriebStetig,		enTypeOfBacNetTextListIn := enTypeOfBacNetTextList.EVENTMESSAGE	),	'E_BI_2_ToOffNormal'	));		
		E_BI_2.IEventMessageTextsConfig.sToFault		:=	fcUtfToAscii(	fcGetBcText(	GVL_BACNET.fbBacNetParameter.metGetTextListName(enTypeOfBacNetFunktionIn := enTypeOfBacNetFunktion.Type_AntriebStetig,		enTypeOfBacNetTextListIn := enTypeOfBacNetTextList.EVENTMESSAGE	),	'E_BI_2_ToFault'		));		
		E_BI_2.IEventMessageTextsConfig.sToNormal		:=	fcUtfToAscii(	fcGetBcText(	GVL_BACNET.fbBacNetParameter.metGetTextListName(enTypeOfBacNetFunktionIn := enTypeOfBacNetFunktion.Type_AntriebStetig,		enTypeOfBacNetTextListIn := enTypeOfBacNetTextList.EVENTMESSAGE	),	'E_BI_2_ToNormal'		));		

		(* Ziel												UTF8->ASCII		BacNet Text		Textlistname									BacNet Funktion																BacNet Textlist type												TextId		*)	
		E_BI_2.sActiveText								:= 	fcUtfToAscii(	fcGetBcText(	GVL_BACNET.fbBacNetParameter.metGetTextListName(enTypeOfBacNetFunktionIn := enTypeOfBacNetFunktion.Type_AntriebStetig,		enTypeOfBacNetTextListIn := enTypeOfBacNetTextList.PRESENTVALUE	),	'E_BI_2_ST_ACTIVE'		));
		E_BI_2.sInactiveText							:= 	fcUtfToAscii(	fcGetBcText(	GVL_BACNET.fbBacNetParameter.metGetTextListName(enTypeOfBacNetFunktionIn := enTypeOfBacNetFunktion.Type_AntriebStetig,		enTypeOfBacNetTextListIn := enTypeOfBacNetTextList.PRESENTVALUE	),	'E_BI_2_ST_INACTIVE'	));	

		(* Ziel												Convert			BacNet Text		Textlistname									BacNet Funktion																BacNet Textlist type												TextId		*)	
		E_BI_2.udiNotificationClass						:= 	TO_UDINT	(	fcGetBcText(	GVL_BACNET.fbBacNetParameter.metGetTextListName(enTypeOfBacNetFunktionIn := enTypeOfBacNetFunktion.Type_AntriebStetig,		enTypeOfBacNetTextListIn := enTypeOfBacNetTextList.NC			),	'E_BI_2_NC'	));	
		E_BI_2.eNotifyType								:= 	WagoTypesBACnet.eBACnetNotifyType.NOTIFY_TYPE_EVENT;
		E_BI_2.xAlarmValue								:= 	TO_BOOL		(	fcGetBcText(	GVL_BACNET.fbBacNetParameter.metGetTextListName(enTypeOfBacNetFunktionIn := enTypeOfBacNetFunktion.Type_AntriebStetig,		enTypeOfBacNetTextListIn := enTypeOfBacNetTextList.NC			),	'E_BI_2_ALV'	));	
		
	ELSE
		E_BI_2.Delete();
	END_IF;
	(* Get Status *)
	metCreate_E_BI_2 := E_BI_2.xIsCreated;	
END_IF;
END_METHOD

METHOD metCreate_B_AI_1 : BOOL
(* B_AI_1*)
IF NOT B_AI_1.xIsCreated THEN
	(* Ziel						UTF8->ASCII						OBJ_NAME_BASE			BacNet Text		Textlistname									BacNet Funktion																BacNet Textlist type												TextId		*)
	B_AI_1._sObjectName		:=	fcUtfToAscii(Standard.CONCAT(	OBJ_NAME_BASE		,	fcGetBcText(	GVL_BACNET.fbBacNetParameter.metGetTextListName(enTypeOfBacNetFunktionIn := enTypeOfBacNetFunktion.Type_AntriebStetig,		enTypeOfBacNetTextListIn := enTypeOfBacNetTextList.ENDING		),	'B_AI_1')));
	B_AI_1._sDescription	:= 	fcUtfToAscii(Standard.CONCAT(	OBJ_NAME_DESCRIPTION,	fcGetBcText(	GVL_BACNET.fbBacNetParameter.metGetTextListName(enTypeOfBacNetFunktionIn := enTypeOfBacNetFunktion.Type_AntriebStetig,		enTypeOfBacNetTextListIn := enTypeOfBacNetTextList.DESCRIPTION	),	'B_AI_1')));
	(* Create Id from Base Id and Object Nr (Last nummber of Name *)	
	B_AI_1.Create(diInstance := TO_DINT(Standard.CONCAT(TO_STRING(dwOBJ_ID_BASE),'1')));
	(* Check if Created *)
	IF B_AI_1.xIsCreated THEN
		(* Set Group *)
		B_AI_1.setPropertyGroup(WagoTypesBacNet.eBACnetPropertyIdentifier.PROP_PRESENT_VALUE						,WagoTypesBacNet.eBACnetPropertyUpdateGroup.GROUP_CYCLIC);
		B_AI_1.setPropertyGroup(WagoTypesBacNet.eBACnetPropertyIdentifier.PROP_PRIORITY_ARRAY						,WagoTypesBacNet.eBACnetPropertyUpdateGroup.GROUP_CYCLIC);
		B_AI_1.setPropertyGroup(WagoTypesBacNet.eBACnetPropertyIdentifier.PROP_ELAPSED_ACTIVE_TIME					,WagoTypesBacNet.eBACnetPropertyUpdateGroup.GROUP_CYCLIC);
		B_AI_1.setPropertyGroup(WagoTypesBacNet.eBACnetPropertyIdentifier.PROP_DESCRIPTION							,WagoTypesBacNet.eBACnetPropertyUpdateGroup.GROUP_CYCLIC);
		B_AI_1.setPropertyGroup(WagoTypesBacNet.eBACnetPropertyIdentifier.PROP_EVENT_MESSAGE_TEXTS_CONFIG			,WagoTypesBacNet.eBACnetPropertyUpdateGroup.GROUP_CYCLIC);
			
		(* Ziel												UTF8->ASCII		BacNet Text		Textlistname									BacNet Funktion																BacNet Textlist type												TextId		*)
		B_AI_1.IEventMessageTextsConfig.sToOffNormal	:=	fcUtfToAscii(	fcGetBcText(	GVL_BACNET.fbBacNetParameter.metGetTextListName(enTypeOfBacNetFunktionIn := enTypeOfBacNetFunktion.Type_AntriebStetig,		enTypeOfBacNetTextListIn := enTypeOfBacNetTextList.EVENTMESSAGE	),	'B_AI_1_ToOffNormal'	));		
		B_AI_1.IEventMessageTextsConfig.sToFault		:=	fcUtfToAscii(	fcGetBcText(	GVL_BACNET.fbBacNetParameter.metGetTextListName(enTypeOfBacNetFunktionIn := enTypeOfBacNetFunktion.Type_AntriebStetig,		enTypeOfBacNetTextListIn := enTypeOfBacNetTextList.EVENTMESSAGE	),	'B_AI_1_ToFault'		));		
		B_AI_1.IEventMessageTextsConfig.sToNormal		:=	fcUtfToAscii(	fcGetBcText(	GVL_BACNET.fbBacNetParameter.metGetTextListName(enTypeOfBacNetFunktionIn := enTypeOfBacNetFunktion.Type_AntriebStetig,		enTypeOfBacNetTextListIn := enTypeOfBacNetTextList.EVENTMESSAGE	),	'B_AI_1_ToNormal'		));		


		(* Ziel												Convert			BacNet Text		Textlistname									BacNet Funktion																BacNet Textlist type												TextId		*)	
		B_AI_1.udiNotificationClass						:= 	TO_UDINT	(	fcGetBcText(	GVL_BACNET.fbBacNetParameter.metGetTextListName(enTypeOfBacNetFunktionIn := enTypeOfBacNetFunktion.Type_AntriebStetig,		enTypeOfBacNetTextListIn := enTypeOfBacNetTextList.NC			),	'B_AI_1_NC'	));	
		B_AI_1.eNotifyType								:= 	WagoTypesBACnet.eBACnetNotifyType.NOTIFY_TYPE_EVENT;
		
	ELSE
		B_AI_1.Delete();
	END_IF;
	(* Get Status *)
	metCreate_B_AI_1 := B_AI_1.xIsCreated;	
END_IF;
END_METHOD

METHOD metCreate_F_BV_1 : BOOL
(* F_BV_1*)
IF NOT F_BV_1.xIsCreated THEN
	(* Ziel						UTF8->ASCII						OBJ_NAME_BASE			BacNet Text		Textlistname									BacNet Funktion																BacNet Textlist type												TextId		*)
	F_BV_1._sObjectName		:=	fcUtfToAscii(Standard.CONCAT(	OBJ_NAME_BASE		,	fcGetBcText(	GVL_BACNET.fbBacNetParameter.metGetTextListName(enTypeOfBacNetFunktionIn := enTypeOfBacNetFunktion.Type_AntriebStetig,		enTypeOfBacNetTextListIn := enTypeOfBacNetTextList.ENDING		),	'F_BV_1')));
	F_BV_1._sDescription	:= 	fcUtfToAscii(Standard.CONCAT(	OBJ_NAME_DESCRIPTION,	fcGetBcText(	GVL_BACNET.fbBacNetParameter.metGetTextListName(enTypeOfBacNetFunktionIn := enTypeOfBacNetFunktion.Type_AntriebStetig,		enTypeOfBacNetTextListIn := enTypeOfBacNetTextList.DESCRIPTION	),	'F_BV_1')));
	(* Create Id from Base Id and Object Nr (Last nummber of Name *)	
	F_BV_1.Create(diInstance := TO_DINT(Standard.CONCAT(TO_STRING(dwOBJ_ID_BASE),'2')));
	(* Check if Created *)
	IF F_BV_1.xIsCreated THEN
		(* Set Group *)
		F_BV_1.setPropertyGroup(WagoTypesBacNet.eBACnetPropertyIdentifier.PROP_PRESENT_VALUE						,WagoTypesBacNet.eBACnetPropertyUpdateGroup.GROUP_CYCLIC);
		F_BV_1.setPropertyGroup(WagoTypesBacNet.eBACnetPropertyIdentifier.PROP_PRIORITY_ARRAY						,WagoTypesBacNet.eBACnetPropertyUpdateGroup.GROUP_CYCLIC);
		F_BV_1.setPropertyGroup(WagoTypesBacNet.eBACnetPropertyIdentifier.PROP_ELAPSED_ACTIVE_TIME					,WagoTypesBacNet.eBACnetPropertyUpdateGroup.GROUP_CYCLIC);
		F_BV_1.setPropertyGroup(WagoTypesBacNet.eBACnetPropertyIdentifier.PROP_DESCRIPTION							,WagoTypesBacNet.eBACnetPropertyUpdateGroup.GROUP_CYCLIC);
		F_BV_1.setPropertyGroup(WagoTypesBacNet.eBACnetPropertyIdentifier.PROP_EVENT_MESSAGE_TEXTS_CONFIG			,WagoTypesBacNet.eBACnetPropertyUpdateGroup.GROUP_CYCLIC);
				
		(* Ziel												UTF8->ASCII		BacNet Text		Textlistname									BacNet Funktion																BacNet Textlist type												TextId		*)
		F_BV_1.IEventMessageTextsConfig.sToOffNormal	:=	fcUtfToAscii(	fcGetBcText(	GVL_BACNET.fbBacNetParameter.metGetTextListName(enTypeOfBacNetFunktionIn := enTypeOfBacNetFunktion.Type_AntriebStetig,		enTypeOfBacNetTextListIn := enTypeOfBacNetTextList.EVENTMESSAGE	),	'F_BV_1_ToOffNormal'	));		
		F_BV_1.IEventMessageTextsConfig.sToFault		:=	fcUtfToAscii(	fcGetBcText(	GVL_BACNET.fbBacNetParameter.metGetTextListName(enTypeOfBacNetFunktionIn := enTypeOfBacNetFunktion.Type_AntriebStetig,		enTypeOfBacNetTextListIn := enTypeOfBacNetTextList.EVENTMESSAGE	),	'F_BV_1_ToFault'		));		
		F_BV_1.IEventMessageTextsConfig.sToNormal		:=	fcUtfToAscii(	fcGetBcText(	GVL_BACNET.fbBacNetParameter.metGetTextListName(enTypeOfBacNetFunktionIn := enTypeOfBacNetFunktion.Type_AntriebStetig,		enTypeOfBacNetTextListIn := enTypeOfBacNetTextList.EVENTMESSAGE	),	'F_BV_1_ToNormal'		));		

		(* Ziel												UTF8->ASCII		BacNet Text		Textlistname									BacNet Funktion																BacNet Textlist type												TextId		*)	
		F_BV_1.sActiveText								:= 	fcUtfToAscii(	fcGetBcText(	GVL_BACNET.fbBacNetParameter.metGetTextListName(enTypeOfBacNetFunktionIn := enTypeOfBacNetFunktion.Type_AntriebStetig,		enTypeOfBacNetTextListIn := enTypeOfBacNetTextList.PRESENTVALUE	),	'F_BV_1_ST_ACTIVE'		));
		F_BV_1.sInactiveText							:= 	fcUtfToAscii(	fcGetBcText(	GVL_BACNET.fbBacNetParameter.metGetTextListName(enTypeOfBacNetFunktionIn := enTypeOfBacNetFunktion.Type_AntriebStetig,		enTypeOfBacNetTextListIn := enTypeOfBacNetTextList.PRESENTVALUE	),	'F_BV_1_ST_INACTIVE'	));	

		(* Ziel												Convert			BacNet Text		Textlistname									BacNet Funktion																BacNet Textlist type												TextId		*)	
		F_BV_1.udiNotificationClass						:= 	TO_UDINT	(	fcGetBcText(	GVL_BACNET.fbBacNetParameter.metGetTextListName(enTypeOfBacNetFunktionIn := enTypeOfBacNetFunktion.Type_AntriebStetig,		enTypeOfBacNetTextListIn := enTypeOfBacNetTextList.NC			),	'F_BV_1_NC'	));	
		F_BV_1.eNotifyType								:= 	WagoTypesBACnet.eBACnetNotifyType.NOTIFY_TYPE_EVENT;
		F_BV_1.xAlarmValue								:= 	TO_BOOL		(	fcGetBcText(	GVL_BACNET.fbBacNetParameter.metGetTextListName(enTypeOfBacNetFunktionIn := enTypeOfBacNetFunktion.Type_AntriebStetig,		enTypeOfBacNetTextListIn := enTypeOfBacNetTextList.NC			),	'F_BV_1_ALV'	));	
		
	ELSE
		F_BV_1.Delete();
	END_IF;
	(* Get Status *)
	metCreate_F_BV_1 := F_BV_1.xIsCreated;	
END_IF;
END_METHOD

METHOD metCREATE_KBOB_2017_V1 : BOOL;
VAR_INPUT
END_VAR
VAR
	oStatus		:	WagoSysErrorBase.FbResult;
	usiErrors	:	USINT;
END_VAR
(* Resett *)
usiErrors := 0;	

(* Create Objeccts *)
CASE usiCreateCase OF
	1:	
		usiErrors := usiErrors + TO_USINT(NOT metCreate_A_AO_1());
	2:
		usiErrors := usiErrors + TO_USINT(NOT metCreate_B_AI_1());
	3:	
		usiErrors := usiErrors + TO_USINT(NOT metCreate_C_TL_1());
	4:	
		usiErrors := usiErrors + TO_USINT(NOT metCreate_D_BI_1());
	5:
		usiErrors := usiErrors + TO_USINT(NOT metCreate_E_BI_2());
	6:	
		usiErrors := usiErrors + TO_USINT(NOT metCreate_F_BV_1());
	0: 
		usiCreateCase := 1;
ELSE
	usiCreateCase := 0;
END_CASE;

(* STRUCT VIEW *)
metCREATE_STRUCTVIEW_KBOB_2017_V1();

(* OK = 0*)
metCREATE_KBOB_2017_V1 := NOT TO_BOOL(usiErrors);
END_METHOD

METHOD metCREATE_STRUCTVIEW_KBOB_2017_V1 : BOOL
VAR_INPUT
END_VAR
CASE usiCreateCase OF
	1:
		fcXMLStructuredView(THIS^,A_AO_1.IObjectIdentifier);
	2:
		fcXMLStructuredView(THIS^,B_AI_1.IObjectIdentifier);
	3:
		fcXMLStructuredView(THIS^,C_TL_1.IObjectIdentifier);
	4:
		fcXMLStructuredView(THIS^,D_BI_1.IObjectIdentifier);
	5:
		fcXMLStructuredView(THIS^,E_BI_2.IObjectIdentifier);
	6:
		fcXMLStructuredView(THIS^,F_BV_1.IObjectIdentifier);
		fcXMLAddStructuredViewToDevice(THIS^);	
	0: 
		usiCreateCase := 1;
ELSE
	usiCreateCase := 0;
END_CASE
END_METHOD

METHOD metCREATE : BOOL;
VAR_INPUT
END_VAR
VAR
	oStatus		:	WagoSysErrorBase.FbResult;
	usiErrors	:	USINT;
END_VAR
(* Get Revision *)
CASE GVL_BACNET.fbBacNetParameter.proKBOB_REV OF
	(* KBOB 2021 V2 *)
	enKBOB_REV.KBOB_REV2021_V2:
		usiErrors := usiErrors + TO_USINT(NOT metCREATE_KBOB_2021_V2());
	(* KBOB 2017 V1 *)
	enKBOB_REV.KBOB_REV2017_V1:
		usiErrors := usiErrors + TO_USINT(NOT metCREATE_KBOB_2017_V1());
	(* Default *)
	ELSE
		usiErrors := usiErrors + TO_USINT(NOT metCREATE_KBOB_2021_V2());
END_CASE;

(* OK = 0*)
xErrorCreate := TO_BOOL(usiErrors);
metCREATE := NOT TO_BOOL(usiErrors) AND usiCreateCase = usiAnzBacNetObj;
END_METHOD

METHOD metCYCLIC_KBOB_2017_V1
VAR_INPUT
END_VAR
(* A_BO_1 *)
IF A_AO_1.IPriorityArray.aLevel[16].xNull OR A_AO_1.IPriorityArray.aLevel[16].rValue <> rRelease THEN
	A_AO_1.IPriorityArray.SetPriority(16,rRelease,FALSE);	// Prio 16 Normal Command
END_IF;
IF xHand THEN
	IF A_AO_1.IPriorityArray.aLevel[7].xNull OR A_AO_1.IPriorityArray.aLevel[7].rValue <> rRelease THEN
		A_AO_1.IPriorityArray.SetPriority(7,rRelease,FALSE);	// Prio 7 Hand Local Command
	END_IF;	
ELSE
	IF NOT A_AO_1.IPriorityArray.aLevel[7].xNull THEN
		A_AO_1.IPriorityArray.SetPriority(7,0,TRUE);			// Prio 7 Hand Local Command NULL
	END_IF;		
END_IF;
IF NOT xSafetyOk THEN
	IF A_AO_1.IPriorityArray.aLevel[5].xNull THEN
		A_AO_1.IPriorityArray.SetPriority( 5,0,FALSE);	// Prio  5 Device safety Off
	END_IF;
ELSE
	IF NOT A_AO_1.IPriorityArray.aLevel[5].xNull THEN
		A_AO_1.IPriorityArray.SetPriority( 5,0,TRUE);	// Prio  5 Device safety NULL
	END_IF;
END_IF;	

(* B_AI_1 *)
IF B_AI_1.rIN <> rAcknowledge THEN
	B_AI_1.rIN := rAcknowledge;
END_IF;

(* D_BI_1 *)
IF D_BI_1.xIN <> xAcknowledgeZu THEN
	D_BI_1.xIN := xAcknowledgeZu;
END_IF;

(* E_BI_2 *)
IF E_BI_2.xIN <> xAcknowledgeAuf THEN
	E_BI_2.xIN := xAcknowledgeAuf;
END_IF;

(* F_BV_1 *)
IF xErrorStellorgan THEN
	IF F_BV_1.IPriorityArray.aLevel[16].xNull THEN
		F_BV_1.IPriorityArray.SetPriority(16,TRUE,FALSE);
	END_IF;
ELSE
	IF NOT F_BV_1.IPriorityArray.aLevel[16].xNull THEN
		F_BV_1.IPriorityArray.SetPriority(16,FALSE,TRUE);
	END_IF;	
END_IF

(* Request Hand Prio 8 *)
xHandPrio8 := NOT A_AO_1.IPriorityArray.aLevel[8].xNull; 
IF xHandPrio8 THEN
	rDemandeHandPrio8 := A_AO_1.IPriorityArray.aLevel[8].rValue;
ELSE
	rDemandeHandPrio8 := 0;
END_IF;
END_METHOD

METHOD metCYCLIC_KBOB_2021_V2
VAR_INPUT
END_VAR
(* A_BO_1 *)
IF A_AO_1.IPriorityArray.aLevel[16].xNull OR A_AO_1.IPriorityArray.aLevel[16].rValue <> rRelease THEN
	A_AO_1.IPriorityArray.SetPriority(16,rRelease,FALSE);	// Prio 16 Normal Command
END_IF;
IF xHand THEN
	IF A_AO_1.IPriorityArray.aLevel[7].xNull OR A_AO_1.IPriorityArray.aLevel[7].rValue <> rRelease THEN
		A_AO_1.IPriorityArray.SetPriority(7,rRelease,FALSE);	// Prio 7 Hand Local Command
	END_IF;	
ELSE
	IF NOT A_AO_1.IPriorityArray.aLevel[7].xNull THEN
		A_AO_1.IPriorityArray.SetPriority(7,0,TRUE);			// Prio 7 Hand Local Command NULL
	END_IF;		
END_IF;
IF NOT xSafetyOk THEN
	IF A_AO_1.IPriorityArray.aLevel[5].xNull THEN
		A_AO_1.IPriorityArray.SetPriority( 5,0,FALSE);	// Prio  5 Device safety Off
	END_IF;
ELSE
	IF NOT A_AO_1.IPriorityArray.aLevel[5].xNull THEN
		A_AO_1.IPriorityArray.SetPriority( 5,0,TRUE);	// Prio  5 Device safety NULL
	END_IF;
END_IF;	

(* B_AI_1 *)
IF B_AI_1.rIN <> rAcknowledge THEN
	B_AI_1.rIN := rAcknowledge;
END_IF;

(* D_BI_1 *)
IF D_BI_1.xIN <> xAcknowledgeZu THEN
	D_BI_1.xIN := xAcknowledgeZu;
END_IF;

(* E_BI_2 *)
IF E_BI_2.xIN <> xAcknowledgeAuf THEN
	E_BI_2.xIN := xAcknowledgeAuf;
END_IF;

(* F_BV_1 *)
IF xErrorStellorgan THEN
	IF F_BV_1.IPriorityArray.aLevel[16].xNull THEN
		F_BV_1.IPriorityArray.SetPriority(16,TRUE,FALSE);
	END_IF;
ELSE
	IF NOT F_BV_1.IPriorityArray.aLevel[16].xNull THEN
		F_BV_1.IPriorityArray.SetPriority(16,FALSE,TRUE);
	END_IF;	
END_IF

(* Request Hand Prio 8 *)
xHandPrio8 := NOT A_AO_1.IPriorityArray.aLevel[8].xNull; 
IF xHandPrio8 THEN
	rDemandeHandPrio8 := A_AO_1.IPriorityArray.aLevel[8].rValue;
ELSE
	rDemandeHandPrio8 := 0;
END_IF;
END_METHOD

METHOD metCYCLIC_DESCRIPTION_FIX
VAR_INPUT
END_VAR
(* A_AO_1 *)
IF A_AO_1.xIsCreated THEN
	IF A_AO_1.sDescription <> A_AO_1._sDescription THEN
		A_AO_1.sDescription := A_AO_1._sDescription;
	END_IF;
END_IF;

(* B_AI_1 *)
IF B_AI_1.xIsCreated THEN
	IF B_AI_1.sDescription <> B_AI_1._sDescription THEN
		B_AI_1.sDescription := B_AI_1._sDescription;
	END_IF;
END_IF;

(* C_TL_1 *)
IF C_TL_1.xIsCreated THEN
	IF C_TL_1.sDescription <> C_TL_1._sDescription THEN
		C_TL_1.sDescription := C_TL_1._sDescription;
	END_IF;
END_IF;

(* D_BI_1 *)
IF D_BI_1.xIsCreated THEN
	IF D_BI_1.sDescription <> D_BI_1._sDescription THEN
		D_BI_1.sDescription := D_BI_1._sDescription;
	END_IF;
END_IF;


(* E_BI_2 *)
IF E_BI_2.xIsCreated THEN
	IF E_BI_2.sDescription <> E_BI_2._sDescription THEN
		E_BI_2.sDescription := E_BI_2._sDescription;
	END_IF;
END_IF;

(* F_BV_1 *)
IF F_BV_1.xIsCreated THEN
	IF F_BV_1.sDescription <> F_BV_1._sDescription THEN
		F_BV_1.sDescription := F_BV_1._sDescription;
	END_IF;
END_IF;
END_METHOD

(*FB_Exit muss explizit implementiert werden. Wenn es eine Implementierung gibt, dann wird 
die Methode aufgerufen, bevor die Steuerung den Code der Funktionsbaustein-Instanz entfernt
(impliziter Aufruf. Der Rückgabewert wird nicht ausgewertet.*)
METHOD FB_Exit : BOOL
VAR_INPUT
	(* TRUE: Die Exit-Methode wird aufgerufen, um die Instanz zu verlassen, die hinterher kopiert wird Online-Change).  *)
	bInCopyCode	: BOOL;
END_VAR
(* A_BO_1*)
IF A_AO_1.xIsCreated THEN
	A_AO_1.Delete();
END_IF;	
(* B_AI_1 *)
IF B_AI_1.xIsCreated THEN
	B_AI_1.Delete();
END_IF;	
(* C_TL_1 *)
IF C_TL_1.xIsCreated THEN
	C_TL_1.Delete();
END_IF;	
(* D_BI_1 *)
IF D_BI_1.xIsCreated THEN
	D_BI_1.Delete();
END_IF;
(* E_BI_2 *)
IF E_BI_2.xIsCreated THEN
	E_BI_2.Delete();
END_IF;
(* F_BV_1 *)
IF F_BV_1.xIsCreated THEN
	F_BV_1.Delete();	
END_IF;
END_METHOD

METHOD metDELETE : BOOL
VAR_INPUT
END_VAR
VAR
	oStatus		:	WagoSysErrorBase.FbResult;
END_VAR
(* A_BO_1*)
IF A_AO_1.xIsCreated THEN
	A_AO_1.Delete(oStatus=>oStatus);
END_IF;	
(* B_AI_1 *)
IF B_AI_1.xIsCreated THEN
	B_AI_1.Delete(oStatus=>oStatus);
END_IF;
(* C_TL_1 *)
IF C_TL_1.xIsCreated THEN
	IF GVL_BACNET.fbBacNetParameter.proDestroyBacNetOverrideXmlNode THEN
		fcXMLDeleteOverrideNode(fcBacNetIdToIdWitType(C_TL_1.IObjectIdentifier.diInstance,C_TL_1.IObjectIdentifier.eObjectType));
	END_IF;
	C_TL_1.Delete(oStatus=>oStatus);
END_IF;	
(* D_BI_1 *)
IF D_BI_1.xIsCreated THEN
	D_BI_1.Delete(oStatus=>oStatus);
END_IF;
(* E_BI_2 *)
IF E_BI_2.xIsCreated THEN
	E_BI_2.Delete(oStatus=>oStatus);
END_IF;
(* F_BV_1 *)
IF F_BV_1.xIsCreated THEN
	F_BV_1.Delete(oStatus=>oStatus);	
END_IF;
(* Delete Struct View *)
IF GVL_BACNET.fbBacNetParameter.proDestroyBacNetOverrideXmlNode THEN
	fcXMLDeleteOverrideNode(fcBacNetIdToIdWitType(TO_DINT(CONCAT(TO_STRING(OBJ_ID_BASE),'1')),WagoTypesBacNet.eBACnetObjectType.BACnet_structured_view));
	fcXMLDeleteStructuredViewFromDevice(fcBacNetIdToIdWitType(TO_DINT(CONCAT(TO_STRING(OBJ_ID_BASE),'1')),WagoTypesBacNet.eBACnetObjectType.BACnet_structured_view));
END_IF;
metDELETE := 	A_AO_1.xIsCreated OR 
				B_AI_1.xIsCreated OR
				C_TL_1.xIsCreated OR				
				D_BI_1.xIsCreated OR
				E_BI_2.xIsCreated OR
				F_BV_1.xIsCreated ;
(* Reset Create Case *)
usiCreateCase := 1;
END_METHOD

END_FUNCTION_BLOCK

// 40 Visualizations/BACNET_PARAMETER/DIA_BACNET_PARAMETER
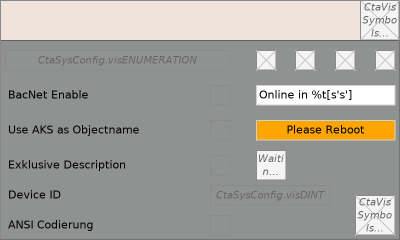
VISUALIZATION DIA_BACNET_PARAMETER  // 400x240
VAR_INPUT
	ITF_BACNET_PARAMETER_IN :	ITF_BACNET_PARAMETER;
END_VAR
    Image (360,0 40x40), image: CtaVisSymbols.ImagePool.close_solo_black
        OnMouseClick:  Dialog=Current Dialog, Result=OK, NumpadKeypadSet=True
    Frame (0,40 400x200), invisible if: NOT __QUERYINTERFACE(ITF_BACNET_PARAMETER_IN,ITF_BACNET_PARAMETER_IN)
        shows VIS_DIA_BACNET_PARAMETER(ITF_BACNET_PARAMETER_IN := ITF_BACNET_PARAMETER_IN)
END_VISUALIZATION

